gfCNCPoint4[21613] = {X 233.3038, Y 9.5049, Z -6.3333, A 0.000, B 0.000, C 0.000 }
gfCNCPoint4[21614] = {X 230.2485, Y 9.5049, Z -6.3333, A 0.000, B 0.000, C 0.000 }
gfCNCPoint4[21615] = {X 230.6107, Y 10.7176, Z -6.3333, A 0.000, B 0.000, C 0.000 }
gfCNCPoint4[21616] = {X 230.7574, Y 11.9748, Z -6.3333, A 0.000, B 0.000, C 0.000 }
gfCNCPoint4[21617] = {X 230.7597, Y 12.0808, Z -6.3333, A 0.000, B 0.000, C 0.000 }
gfCNCPoint4[21618] = {X 230.7605, Y 12.1868, Z -6.3333, A 0.000, B 0.000, C 0.000 }
gfCNCPoint4[21619] = {X 230.7602, Y 13.0462, Z -6.3333, A 0.000, B 0.000, C 0.000 }
gfCNCPoint4[21620] = {X 230.6532, Y 14.2233, Z -6.3333, A 0.000, B 0.000, C 0.000 }
gfCNCPoint4[21621] = {X 230.3572, Y 15.3675, Z -6.3333, A 0.000, B 0.000, C 0.000 }
gfCNCPoint4[21622] = {X 229.8799, Y 16.4488, Z -6.3333, A 0.000, B 0.000, C 0.000 }
gfCNCPoint4[21623] = {X 229.2339, Y 17.4386, Z -6.3333, A 0.000, B 0.000, C 0.000 }
gfCNCPoint4[21624] = {X 229.2342, Y 25.8570, Z -6.3333, A 0.000, B 0.000, C 0.000 }
gfCNCPoint4[21625] = {X 231.6342, Y 25.8569, Z -6.3333, A 0.000, B 0.000, C 0.000 }
gfCNCPoint4[21626] = {X 231.6347, Y 38.9924, Z -6.3333, A 0.000, B 0.000, C 0.000 }
gfCNCPoint4[21627] = {X 231.6440, Y 39.0069, Z -6.3333, A 0.000, B 0.000, C 0.000 }
gfCNCPoint4[21628] = {X 232.3931, Y 37.9855, Z -6.3333, A 0.000, B 0.000, C 0.000 }
gfCNCPoint4[21629] = {X 233.2692, Y 37.0706, Z -6.3333, A 0.000, B 0.000, C 0.000 }
gfCNCPoint4[21630] = {X 234.2573, Y 36.2780, Z -6.3333, A 0.000, B 0.000, C 0.000 }
gfCNCPoint4[21631] = {X 235.5691, Y 33.7103, Z -6.3333, A 0.000, B 0.000, C 0.000 }
gfCNCPoint4[21632] = {X 234.4282, Y 32.2860, Z -6.3333, A 0.000, B 0.000, C 0.000 }
gfCNCPoint4[21633] = {X 233.4498, Y 30.7456, Z -6.3333, A 0.000, B 0.000, C 0.000 }
gfCNCPoint4[21634] = {X 232.6455, Y 29.1076, Z -6.3333, A 0.000, B 0.000, C 0.000 }
gfCNCPoint4[21635] = {X 232.0249, Y 27.3915, Z -6.3333, A 0.000, B 0.000, C 0.000 }
gfCNCPoint4[21636] = {X 231.8157, Y 26.6277, Z -6.3333, A 0.000, B 0.000, C 0.000 }
gfCNCPoint4[21637] = {X 231.6342, Y 25.8569, Z -6.3333, A 0.000, B 0.000, C 0.000 }
gfCNCPoint4[21638] = {X 229.2342, Y 25.8570, Z -6.3333, A 0.000, B 0.000, C 0.000 }
gfCNCPoint4[21639] = {X 229.2347, Y 39.7493, Z -6.3333, A 0.000, B 0.000, C 0.000 }
gfCNCPoint4[21640] = {X 229.4337, Y 40.0185, Z -6.3333, A 0.000, B 0.000, C 0.000 }
gfCNCPoint4[21641] = {X 229.6200, Y 40.2966, Z -6.3333, A 0.000, B 0.000, C 0.000 }
gfCNCPoint4[21642] = {X 230.1055, Y 41.1910, Z -6.3333, A 0.000, B 0.000, C 0.000 }
gfCNCPoint4[21643] = {X 230.4616, Y 42.1443, Z -6.3333, A 0.000, B 0.000, C 0.000 }
gfCNCPoint4[21644] = {X 230.6813, Y 43.1379, Z -6.3333, A 0.000, B 0.000, C 0.000 }
gfCNCPoint4[21645] = {X 230.7603, Y 44.1524, Z -6.3333, A 0.000, B 0.000, C 0.000 }
gfCNCPoint4[21646] = {X 230.7605, Y 45.0000, Z -6.3333, A 0.000, B 0.000, C 0.000 }
gfCNCPoint4[21647] = {X 230.7459, Y 45.4609, Z -6.3333, A 0.000, B 0.000, C 0.000 }
gfCNCPoint4[21648] = {X 230.7021, Y 45.9200, Z -6.3333, A 0.000, B 0.000, C 0.000 }
gfCNCPoint4[21649] = {X 232.5859, Y 45.9200, Z -6.3333, A 0.000, B 0.000, C 0.000 }
gfCNCPoint4[21650] = {X 232.5421, Y 45.4609, Z -6.3333, A 0.000, B 0.000, C 0.000 }
gfCNCPoint4[21651] = {X 232.5275, Y 45.0000, Z -6.3333, A 0.000, B 0.000, C 0.000 }
gfCNCPoint4[21652] = {X 232.5275, Y 44.2089, Z -6.3333, A 0.000, B 0.000, C 0.000 }
gfCNCPoint4[21653] = {X 232.6006, Y 43.1798, Z -6.3333, A 0.000, B 0.000, C 0.000 }
gfCNCPoint4[21654] = {X 232.8184, Y 42.1714, Z -6.3333, A 0.000, B 0.000, C 0.000 }
gfCNCPoint4[21655] = {X 233.1766, Y 41.2038, Z -6.3333, A 0.000, B 0.000, C 0.000 }
gfCNCPoint4[21656] = {X 233.6680, Y 40.2966, Z -6.3333, A 0.000, B 0.000, C 0.000 }
gfCNCPoint4[21657] = {X 234.3527, Y 39.3876, Z -6.3333, A 0.000, B 0.000, C 0.000 }
gfCNCPoint4[21658] = {X 235.1707, Y 38.5964, Z -6.3333, A 0.000, B 0.000, C 0.000 }
gfCNCPoint4[21659] = {X 236.1021, Y 37.9424, Z -6.3333, A 0.000, B 0.000, C 0.000 }
gfCNCPoint4[21660] = {X 238.4997, Y 33.2492, Z -6.3333, A 0.000, B 0.000, C 0.000 }
gfCNCPoint4[21661] = {X 237.3859, Y 32.1414, Z -6.3333, A 0.000, B 0.000, C 0.000 }
gfCNCPoint4[21662] = {X 236.4005, Y 30.9179, Z -6.3333, A 0.000, B 0.000, C 0.000 }
gfCNCPoint4[21663] = {X 235.5554, Y 29.5936, Z -6.3333, A 0.000, B 0.000, C 0.000 }
gfCNCPoint4[21664] = {X 234.8609, Y 28.1845, Z -6.3333, A 0.000, B 0.000, C 0.000 }
gfCNCPoint4[21665] = {X 234.3254, Y 26.7076, Z -6.3333, A 0.000, B 0.000, C 0.000 }
gfCNCPoint4[21666] = {X 234.1405, Y 26.0316, Z -6.3333, A 0.000, B 0.000, C 0.000 }
gfCNCPoint4[21667] = {X 233.9799, Y 25.3493, Z -6.3333, A 0.000, B 0.000, C 0.000 }
gfCNCPoint4[21668] = {X 233.6672, Y 23.4597, Z -6.3333, A 0.000, B 0.000, C 0.000 }
gfCNCPoint4[21669] = {X 233.5414, Y 21.5485, Z -6.3333, A 0.000, B 0.000, C 0.000 }
gfCNCPoint4[21670] = {X 233.6038, Y 19.6342, Z -6.3333, A 0.000, B 0.000, C 0.000 }
gfCNCPoint4[21671] = {X 233.8537, Y 17.7353, Z -6.3333, A 0.000, B 0.000, C 0.000 }
gfCNCPoint4[21672] = {X 234.2887, Y 15.8701, Z -6.3333, A 0.000, B 0.000, C 0.000 }
gfCNCPoint4[21673] = {X 234.7349, Y 14.5420, Z -6.3333, A 0.000, B 0.000, C 0.000 }
gfCNCPoint4[21674] = {X 235.3045, Y 13.2620, Z -6.3333, A 0.000, B 0.000, C 0.000 }
gfCNCPoint4[21675] = {X 235.3657, Y 13.1418, Z -6.3333, A 0.000, B 0.000, C 0.000 }
gfCNCPoint4[21676] = {X 235.4279, Y 13.0222, Z -6.3333, A 0.000, B 0.000, C 0.000 }
gfCNCPoint4[21677] = {X 236.1692, Y 11.7670, Z -6.3333, A 0.000, B 0.000, C 0.000 }
gfCNCPoint4[21678] = {X 237.0303, Y 10.5908, Z -6.3333, A 0.000, B 0.000, C 0.000 }
gfCNCPoint4[21679] = {X 238.0029, Y 9.5049, Z -6.3333, A 0.000, B 0.000, C 0.000 }
gfCNCPoint4[21680] = {X 233.3038, Y 9.5049, Z -6.3333, A 0.000, B 0.000, C 0.000 }
gfCNCPoint4[21681] = {X 233.3038, Y 7.1049, Z -6.3333, A 0.000, B 0.000, C 0.000 }
gfCNCPoint4[21682] = {X 207.3611, Y 7.1049, Z -6.3333, A 0.000, B 0.000, C 0.000 }
gfCNCPoint4[21683] = {X 207.3611, Y 11.9049, Z -6.3333, A 0.000, B 0.000, C 0.000 }
gfCNCPoint4[21684] = {X 205.8579, Y 11.9049, Z -6.3333, A 0.000, B 0.000, C 0.000 }
gfCNCPoint4[21685] = {X 206.6129, Y 13.3419, Z -6.3333, A 0.000, B 0.000, C 0.000 }
gfCNCPoint4[21686] = {X 207.2383, Y 14.8398, Z -6.3333, A 0.000, B 0.000, C 0.000 }
gfCNCPoint4[21687] = {X 207.7991, Y 16.7126, Z -6.3333, A 0.000, B 0.000, C 0.000 }
gfCNCPoint4[21688] = {X 208.1779, Y 18.6305, Z -6.3333, A 0.000, B 0.000, C 0.000 }
gfCNCPoint4[21689] = {X 208.3712, Y 20.5759, Z -6.3333, A 0.000, B 0.000, C 0.000 }
gfCNCPoint4[21690] = {X 208.3773, Y 22.5308, Z -6.3333, A 0.000, B 0.000, C 0.000 }
gfCNCPoint4[21691] = {X 208.1960, Y 24.4773, Z -6.3333, A 0.000, B 0.000, C 0.000 }
gfCNCPoint4[21692] = {X 207.8292, Y 26.3975, Z -6.3333, A 0.000, B 0.000, C 0.000 }
gfCNCPoint4[21693] = {X 207.3620, Y 28.0101, Z -6.3333, A 0.000, B 0.000, C 0.000 }
gfCNCPoint4[21694] = {X 206.7385, Y 29.5690, Z -6.3333, A 0.000, B 0.000, C 0.000 }
gfCNCPoint4[21695] = {X 205.9648, Y 31.0590, Z -6.3333, A 0.000, B 0.000, C 0.000 }
gfCNCPoint4[21696] = {X 206.0466, Y 31.2168, Z -6.3333, A 0.000, B 0.000, C 0.000 }
gfCNCPoint4[21697] = {X 206.1255, Y 31.3760, Z -6.3333, A 0.000, B 0.000, C 0.000 }
gfCNCPoint4[21698] = {X 208.8842, Y 37.0755, Z -6.3333, A 0.000, B 0.000, C 0.000 }
gfCNCPoint4[21699] = {X 208.8842, Y 18.1966, Z -6.3333, A 0.000, B 0.000, C 0.000 }
gfCNCPoint4[21700] = {X 208.2325, Y 17.0008, Z -6.3333, A 0.000, B 0.000, C 0.000 }
gfCNCPoint4[21701] = {X 207.7551, Y 15.7254, Z -6.3333, A 0.000, B 0.000, C 0.000 }
gfCNCPoint4[21702] = {X 207.4614, Y 14.3956, Z -6.3333, A 0.000, B 0.000, C 0.000 }
gfCNCPoint4[21703] = {X 207.3572, Y 13.0378, Z -6.3333, A 0.000, B 0.000, C 0.000 }
gfCNCPoint4[21704] = {X 207.3570, Y 12.1868, Z -6.3333, A 0.000, B 0.000, C 0.000 }
gfCNCPoint4[21705] = {X 207.3580, Y 12.0458, Z -6.3333, A 0.000, B 0.000, C 0.000 }
gfCNCPoint4[21706] = {X 207.3611, Y 11.9049, Z -6.3333, A 0.000, B 0.000, C 0.000 }
gfCNCPoint4[21707] = {X 207.3611, Y 9.5049, Z -6.3333, A 0.000, B 0.000, C 0.000 }
gfCNCPoint4[21708] = {X 200.9085, Y 9.5049, Z -6.3333, A 0.000, B 0.000, C 0.000 }
gfCNCPoint4[21709] = {X 201.9821, Y 10.6133, Z -6.3333, A 0.000, B 0.000, C 0.000 }
gfCNCPoint4[21710] = {X 202.9438, Y 11.8201, Z -6.3333, A 0.000, B 0.000, C 0.000 }
gfCNCPoint4[21711] = {X 203.7847, Y 13.1140, Z -6.3333, A 0.000, B 0.000, C 0.000 }
gfCNCPoint4[21712] = {X 204.4380, Y 14.3567, Z -6.3333, A 0.000, B 0.000, C 0.000 }
gfCNCPoint4[21713] = {X 204.9798, Y 15.6519, Z -6.3333, A 0.000, B 0.000, C 0.000 }
gfCNCPoint4[21714] = {X 205.5523, Y 17.6384, Z -6.3333, A 0.000, B 0.000, C 0.000 }
gfCNCPoint4[21715] = {X 205.8929, Y 19.6775, Z -6.3333, A 0.000, B 0.000, C 0.000 }
gfCNCPoint4[21716] = {X 205.9974, Y 21.7422, Z -6.3333, A 0.000, B 0.000, C 0.000 }
gfCNCPoint4[21717] = {X 205.8641, Y 23.8052, Z -6.3333, A 0.000, B 0.000, C 0.000 }
gfCNCPoint4[21718] = {X 205.4950, Y 25.8393, Z -6.3333, A 0.000, B 0.000, C 0.000 }
gfCNCPoint4[21719] = {X 205.0938, Y 27.2257, Z -6.3333, A 0.000, B 0.000, C 0.000 }
gfCNCPoint4[21720] = {X 204.5582, Y 28.5659, Z -6.3333, A 0.000, B 0.000, C 0.000 }
gfCNCPoint4[21721] = {X 203.8933, Y 29.8469, Z -6.3333, A 0.000, B 0.000, C 0.000 }
gfCNCPoint4[21722] = {X 203.1057, Y 31.0563, Z -6.3333, A 0.000, B 0.000, C 0.000 }
gfCNCPoint4[21723] = {X 203.5734, Y 31.7151, Z -6.3333, A 0.000, B 0.000, C 0.000 }
gfCNCPoint4[21724] = {X 203.9653, Y 32.4217, Z -6.3333, A 0.000, B 0.000, C 0.000 }
gfCNCPoint4[21725] = {X 206.9865, Y 38.6634, Z -6.3333, A 0.000, B 0.000, C 0.000 }
gfCNCPoint4[21726] = {X 207.4240, Y 39.8017, Z -6.3333, A 0.000, B 0.000, C 0.000 }
gfCNCPoint4[21727] = {X 207.6653, Y 40.9971, Z -6.3333, A 0.000, B 0.000, C 0.000 }
gfCNCPoint4[21728] = {X 207.7038, Y 42.2159, Z -6.3333, A 0.000, B 0.000, C 0.000 }
gfCNCPoint4[21729] = {X 207.5382, Y 43.4241, Z -6.3333, A 0.000, B 0.000, C 0.000 }
gfCNCPoint4[21730] = {X 207.1733, Y 44.5877, Z -6.3333, A 0.000, B 0.000, C 0.000 }
gfCNCPoint4[21731] = {X 206.6193, Y 45.6741, Z -6.3333, A 0.000, B 0.000, C 0.000 }
gfCNCPoint4[21732] = {X 205.8917, Y 46.6527, Z -6.3333, A 0.000, B 0.000, C 0.000 }
gfCNCPoint4[21733] = {X 205.0110, Y 47.4962, Z -6.3333, A 0.000, B 0.000, C 0.000 }
gfCNCPoint4[21734] = {X 204.4751, Y 47.9295, Z -6.3333, A 0.000, B 0.000, C 0.000 }
gfCNCPoint4[21735] = {X 203.5896, Y 48.5433, Z -6.3333, A 0.000, B 0.000, C 0.000 }
gfCNCPoint4[21736] = {X 202.6234, Y 49.0199, Z -6.3333, A 0.000, B 0.000, C 0.000 }
gfCNCPoint4[21737] = {X 201.4894, Y 49.3740, Z -6.3333, A 0.000, B 0.000, C 0.000 }
gfCNCPoint4[21738] = {X 200.3130, Y 49.5392, Z -6.3333, A 0.000, B 0.000, C 0.000 }
gfCNCPoint4[21739] = {X 199.1253, Y 49.5112, Z -6.3333, A 0.000, B 0.000, C 0.000 }
gfCNCPoint4[21740] = {X 197.0993, Y 50.4925, Z -6.3333, A 0.000, B 0.000, C 0.000 }
gfCNCPoint4[21741] = {X 195.0081, Y 51.3261, Z -6.3333, A 0.000, B 0.000, C 0.000 }
gfCNCPoint4[21742] = {X 192.8625, Y 52.0075, Z -6.3333, A 0.000, B 0.000, C 0.000 }
gfCNCPoint4[21743] = {X 192.4425, Y 52.1234, Z -6.3333, A 0.000, B 0.000, C 0.000 }
gfCNCPoint4[21744] = {X 192.0206, Y 52.2321, Z -6.3333, A 0.000, B 0.000, C 0.000 }
gfCNCPoint4[21745] = {X 190.7204, Y 52.5192, Z -6.3333, A 0.000, B 0.000, C 0.000 }
gfCNCPoint4[21746] = {X 189.4070, Y 52.7376, Z -6.3333, A 0.000, B 0.000, C 0.000 }
gfCNCPoint4[21747] = {X 189.9007, Y 53.9117, Z -6.3333, A 0.000, B 0.000, C 0.000 }
gfCNCPoint4[21748] = {X 190.2679, Y 55.1313, Z -6.3333, A 0.000, B 0.000, C 0.000 }
gfCNCPoint4[21749] = {X 190.5268, Y 56.5553, Z -6.3333, A 0.000, B 0.000, C 0.000 }
gfCNCPoint4[21750] = {X 190.6135, Y 58.0000, Z -6.3333, A 0.000, B 0.000, C 0.000 }
gfCNCPoint4[21751] = {X 190.6132, Y 58.8756, Z -6.3333, A 0.000, B 0.000, C 0.000 }
gfCNCPoint4[21752] = {X 208.6248, Y 78.5343, Z -6.3333, A 0.000, B 0.000, C 0.000 }
gfCNCPoint4[21753] = {X 212.1639, Y 75.2917, Z -6.3333, A 0.000, B 0.000, C 0.000 }
gfCNCPoint4[21754] = {X 215.1986, Y 78.6038, Z -6.3333, A 0.000, B 0.000, C 0.000 }
gfCNCPoint4[21755] = {X 218.3263, Y 76.6002, Z -6.3333, A 0.000, B 0.000, C 0.000 }
gfCNCPoint4[21756] = {X 216.9980, Y 76.0790, Z -6.3333, A 0.000, B 0.000, C 0.000 }
gfCNCPoint4[21757] = {X 216.3745, Y 75.8855, Z -6.3333, A 0.000, B 0.000, C 0.000 }
gfCNCPoint4[21758] = {X 215.7268, Y 75.8033, Z -6.3333, A 0.000, B 0.000, C 0.000 }
gfCNCPoint4[21759] = {X 213.9317, Y 75.6427, Z -6.3333, A 0.000, B 0.000, C 0.000 }
gfCNCPoint4[21760] = {X 212.1639, Y 75.2917, Z -6.3333, A 0.000, B 0.000, C 0.000 }
gfCNCPoint4[21761] = {X 210.3944, Y 76.9130, Z -6.3333, A 0.000, B 0.000, C 0.000 }
gfCNCPoint4[21762] = {X 214.7930, Y 81.7139, Z -6.3333, A 0.000, B 0.000, C 0.000 }
gfCNCPoint4[21763] = {X 223.5811, Y 76.0841, Z -6.3333, A 0.000, B 0.000, C 0.000 }
gfCNCPoint4[21764] = {X 217.8868, Y 73.8496, Z -6.3333, A 0.000, B 0.000, C 0.000 }
gfCNCPoint4[21765] = {X 216.8707, Y 73.5373, Z -6.3333, A 0.000, B 0.000, C 0.000 }
gfCNCPoint4[21766] = {X 215.8159, Y 73.4049, Z -6.3333, A 0.000, B 0.000, C 0.000 }
gfCNCPoint4[21767] = {X 214.2744, Y 73.2673, Z -6.3333, A 0.000, B 0.000, C 0.000 }
gfCNCPoint4[21768] = {X 212.7564, Y 72.9660, Z -6.3333, A 0.000, B 0.000, C 0.000 }
gfCNCPoint4[21769] = {X 211.1573, Y 72.4583, Z -6.3333, A 0.000, B 0.000, C 0.000 }
gfCNCPoint4[21770] = {X 209.6276, Y 71.7691, Z -6.3333, A 0.000, B 0.000, C 0.000 }
gfCNCPoint4[21771] = {X 208.1879, Y 70.9075, Z -6.3333, A 0.000, B 0.000, C 0.000 }
gfCNCPoint4[21772] = {X 206.8576, Y 69.8853, Z -6.3333, A 0.000, B 0.000, C 0.000 }
gfCNCPoint4[21773] = {X 205.6544, Y 68.7159, Z -6.3333, A 0.000, B 0.000, C 0.000 }
gfCNCPoint4[21774] = {X 204.5946, Y 67.4153, Z -6.3333, A 0.000, B 0.000, C 0.000 }
gfCNCPoint4[21775] = {X 203.6923, Y 66.0008, Z -6.3333, A 0.000, B 0.000, C 0.000 }
gfCNCPoint4[21776] = {X 202.9597, Y 64.4914, Z -6.3333, A 0.000, B 0.000, C 0.000 }
gfCNCPoint4[21777] = {X 202.4066, Y 62.9075, Z -6.3333, A 0.000, B 0.000, C 0.000 }
gfCNCPoint4[21778] = {X 202.0405, Y 61.2701, Z -6.3333, A 0.000, B 0.000, C 0.000 }
gfCNCPoint4[21779] = {X 199.6719, Y 61.6573, Z -6.3333, A 0.000, B 0.000, C 0.000 }
gfCNCPoint4[21780] = {X 199.5094, Y 60.3398, Z -6.3333, A 0.000, B 0.000, C 0.000 }
gfCNCPoint4[21781] = {X 199.4510, Y 59.0136, Z -6.3333, A 0.000, B 0.000, C 0.000 }
gfCNCPoint4[21782] = {X 199.4508, Y 58.0000, Z -6.3333, A 0.000, B 0.000, C 0.000 }
gfCNCPoint4[21783] = {X 199.5411, Y 56.2566, Z -6.3333, A 0.000, B 0.000, C 0.000 }
gfCNCPoint4[21784] = {X 199.8109, Y 54.5319, Z -6.3333, A 0.000, B 0.000, C 0.000 }
gfCNCPoint4[21785] = {X 197.5976, Y 55.4819, Z -6.3333, A 0.000, B 0.000, C 0.000 }
gfCNCPoint4[21786] = {X 195.3259, Y 56.2825, Z -6.3333, A 0.000, B 0.000, C 0.000 }
gfCNCPoint4[21787] = {X 195.3577, Y 56.6287, Z -6.3333, A 0.000, B 0.000, C 0.000 }
gfCNCPoint4[21788] = {X 195.3824, Y 56.9755, Z -6.3333, A 0.000, B 0.000, C 0.000 }
gfCNCPoint4[21789] = {X 199.6719, Y 61.6573, Z -6.3333, A 0.000, B 0.000, C 0.000 }
gfCNCPoint4[21790] = {X 202.0405, Y 61.2701, Z -6.3333, A 0.000, B 0.000, C 0.000 }
gfCNCPoint4[21791] = {X 201.9013, Y 60.1424, Z -6.3333, A 0.000, B 0.000, C 0.000 }
gfCNCPoint4[21792] = {X 201.8510, Y 59.0073, Z -6.3333, A 0.000, B 0.000, C 0.000 }
gfCNCPoint4[21793] = {X 201.8508, Y 58.0000, Z -6.3333, A 0.000, B 0.000, C 0.000 }
gfCNCPoint4[21794] = {X 201.9282, Y 56.5045, Z -6.3333, A 0.000, B 0.000, C 0.000 }
gfCNCPoint4[21795] = {X 202.1597, Y 55.0250, Z -6.3333, A 0.000, B 0.000, C 0.000 }
gfCNCPoint4[21796] = {X 202.4964, Y 53.7245, Z -6.3333, A 0.000, B 0.000, C 0.000 }
gfCNCPoint4[21797] = {X 202.9522, Y 52.4609, Z -6.3333, A 0.000, B 0.000, C 0.000 }
gfCNCPoint4[21798] = {X 203.5231, Y 51.2449, Z -6.3333, A 0.000, B 0.000, C 0.000 }
gfCNCPoint4[21799] = {X 202.2638, Y 51.6564, Z -6.3333, A 0.000, B 0.000, C 0.000 }
gfCNCPoint4[21800] = {X 200.9603, Y 51.8923, Z -6.3333, A 0.000, B 0.000, C 0.000 }
gfCNCPoint4[21801] = {X 199.6367, Y 51.9482, Z -6.3333, A 0.000, B 0.000, C 0.000 }
gfCNCPoint4[21802] = {X 199.2155, Y 52.1566, Z -6.3333, A 0.000, B 0.000, C 0.000 }
gfCNCPoint4[21803] = {X 198.7914, Y 52.3592, Z -6.3333, A 0.000, B 0.000, C 0.000 }
gfCNCPoint4[21804] = {X 196.1934, Y 53.4485, Z -6.3333, A 0.000, B 0.000, C 0.000 }
gfCNCPoint4[21805] = {X 193.5136, Y 54.3175, Z -6.3333, A 0.000, B 0.000, C 0.000 }
gfCNCPoint4[21806] = {X 193.0575, Y 54.4433, Z -6.3333, A 0.000, B 0.000, C 0.000 }
gfCNCPoint4[21807] = {X 192.5993, Y 54.5613, Z -6.3333, A 0.000, B 0.000, C 0.000 }
gfCNCPoint4[21808] = {X 192.9061, Y 56.2397, Z -6.3333, A 0.000, B 0.000, C 0.000 }
gfCNCPoint4[21809] = {X 193.0134, Y 57.9426, Z -6.3333, A 0.000, B 0.000, C 0.000 }
gfCNCPoint4[21810] = {X 210.3944, Y 76.9130, Z -6.3333, A 0.000, B 0.000, C 0.000 }
gfCNCPoint4[21811] = {X 208.6248, Y 78.5343, Z -6.3333, A 0.000, B 0.000, C 0.000 }
gfCNCPoint4[21812] = {X 214.3875, Y 84.8240, Z -6.3333, A 0.000, B 0.000, C 0.000 }
gfCNCPoint4[21813] = {X 228.8358, Y 75.5680, Z -6.3333, A 0.000, B 0.000, C 0.000 }
gfCNCPoint4[21814] = {X 218.7736, Y 71.6194, Z -6.3333, A 0.000, B 0.000, C 0.000 }
gfCNCPoint4[21815] = {X 217.8428, Y 71.3053, Z -6.3333, A 0.000, B 0.000, C 0.000 }
gfCNCPoint4[21816] = {X 216.8820, Y 71.1001, Z -6.3333, A 0.000, B 0.000, C 0.000 }
gfCNCPoint4[21817] = {X 215.9041, Y 71.0065, Z -6.3333, A 0.000, B 0.000, C 0.000 }
gfCNCPoint4[21818] = {X 214.2345, Y 70.8308, Z -6.3333, A 0.000, B 0.000, C 0.000 }
gfCNCPoint4[21819] = {X 212.6054, Y 70.4253, Z -6.3333, A 0.000, B 0.000, C 0.000 }
gfCNCPoint4[21820] = {X 211.0482, Y 69.7978, Z -6.3333, A 0.000, B 0.000, C 0.000 }
gfCNCPoint4[21821] = {X 209.5931, Y 68.9605, Z -6.3333, A 0.000, B 0.000, C 0.000 }
gfCNCPoint4[21822] = {X 208.2681, Y 67.9296, Z -6.3333, A 0.000, B 0.000, C 0.000 }
gfCNCPoint4[21823] = {X 207.0988, Y 66.7249, Z -6.3333, A 0.000, B 0.000, C 0.000 }
gfCNCPoint4[21824] = {X 206.1079, Y 65.3697, Z -6.3333, A 0.000, B 0.000, C 0.000 }
gfCNCPoint4[21825] = {X 205.3143, Y 63.8903, Z -6.3333, A 0.000, B 0.000, C 0.000 }
gfCNCPoint4[21826] = {X 204.7336, Y 62.3151, Z -6.3333, A 0.000, B 0.000, C 0.000 }
gfCNCPoint4[21827] = {X 204.3768, Y 60.6746, Z -6.3333, A 0.000, B 0.000, C 0.000 }
gfCNCPoint4[21828] = {X 204.2510, Y 59.0005, Z -6.3333, A 0.000, B 0.000, C 0.000 }
gfCNCPoint4[21829] = {X 204.2508, Y 58.0000, Z -6.3333, A 0.000, B 0.000, C 0.000 }
gfCNCPoint4[21830] = {X 204.3396, Y 56.5378, Z -6.3333, A 0.000, B 0.000, C 0.000 }
gfCNCPoint4[21831] = {X 204.6048, Y 55.0972, Z -6.3333, A 0.000, B 0.000, C 0.000 }
gfCNCPoint4[21832] = {X 205.0423, Y 53.6992, Z -6.3333, A 0.000, B 0.000, C 0.000 }
gfCNCPoint4[21833] = {X 205.6459, Y 52.3645, Z -6.3333, A 0.000, B 0.000, C 0.000 }
gfCNCPoint4[21834] = {X 206.5294, Y 50.9389, Z -6.3333, A 0.000, B 0.000, C 0.000 }
gfCNCPoint4[21835] = {X 207.6019, Y 49.6494, Z -6.3333, A 0.000, B 0.000, C 0.000 }
gfCNCPoint4[21836] = {X 208.8426, Y 48.5209, Z -6.3333, A 0.000, B 0.000, C 0.000 }
gfCNCPoint4[21837] = {X 210.2277, Y 47.5751, Z -6.3333, A 0.000, B 0.000, C 0.000 }
gfCNCPoint4[21838] = {X 209.8801, Y 46.3328, Z -6.3333, A 0.000, B 0.000, C 0.000 }
gfCNCPoint4[21839] = {X 209.7572, Y 45.0487, Z -6.3333, A 0.000, B 0.000, C 0.000 }
gfCNCPoint4[21840] = {X 209.7570, Y 44.1918, Z -6.3333, A 0.000, B 0.000, C 0.000 }
gfCNCPoint4[21841] = {X 209.8558, Y 43.0029, Z -6.3333, A 0.000, B 0.000, C 0.000 }
gfCNCPoint4[21842] = {X 210.1495, Y 41.8467, Z -6.3333, A 0.000, B 0.000, C 0.000 }
gfCNCPoint4[21843] = {X 210.6300, Y 40.7548, Z -6.3333, A 0.000, B 0.000, C 0.000 }
gfCNCPoint4[21844] = {X 211.2842, Y 39.7572, Z -6.3333, A 0.000, B 0.000, C 0.000 }
gfCNCPoint4[21845] = {X 211.2842, Y 37.0755, Z -6.3333, A 0.000, B 0.000, C 0.000 }
gfCNCPoint4[21846] = {X 211.2839, Y 17.4390, Z -6.3333, A 0.000, B 0.000, C 0.000 }
gfCNCPoint4[21847] = {X 210.6358, Y 16.4454, Z -6.3333, A 0.000, B 0.000, C 0.000 }
gfCNCPoint4[21848] = {X 210.1576, Y 15.3597, Z -6.3333, A 0.000, B 0.000, C 0.000 }
gfCNCPoint4[21849] = {X 209.8621, Y 14.2108, Z -6.3333, A 0.000, B 0.000, C 0.000 }
gfCNCPoint4[21850] = {X 209.7572, Y 13.0291, Z -6.3333, A 0.000, B 0.000, C 0.000 }
gfCNCPoint4[21851] = {X 209.7570, Y 12.1868, Z -6.3333, A 0.000, B 0.000, C 0.000 }
gfCNCPoint4[21852] = {X 209.7578, Y 12.0808, Z -6.3333, A 0.000, B 0.000, C 0.000 }
gfCNCPoint4[21853] = {X 209.7601, Y 11.9748, Z -6.3333, A 0.000, B 0.000, C 0.000 }
gfCNCPoint4[21854] = {X 209.9068, Y 10.7176, Z -6.3333, A 0.000, B 0.000, C 0.000 }
gfCNCPoint4[21855] = {X 210.2690, Y 9.5049, Z -6.3333, A 0.000, B 0.000, C 0.000 }
gfCNCPoint4[21856] = {X 207.3611, Y 9.5049, Z -6.3333, A 0.000, B 0.000, C 0.000 }
gfCNCPoint4[21857] = {X 207.3611, Y 7.1049, Z -6.3333, A 0.000, B 0.000, C 0.000 }
gfCNCPoint4[21858] = {X 191.0955, Y 7.1049, Z -6.3333, A 0.000, B 0.000, C 0.000 }
gfCNCPoint4[21859] = {X 193.0686, Y 7.6379, Z -6.3333, A 0.000, B 0.000, C 0.000 }
gfCNCPoint4[21860] = {X 194.9670, Y 8.3953, Z -6.3333, A 0.000, B 0.000, C 0.000 }
gfCNCPoint4[21861] = {X 196.7651, Y 9.3670, Z -6.3333, A 0.000, B 0.000, C 0.000 }
gfCNCPoint4[21862] = {X 198.4389, Y 10.5400, Z -6.3333, A 0.000, B 0.000, C 0.000 }
gfCNCPoint4[21863] = {X 198.8603, Y 10.8896, Z -6.3333, A 0.000, B 0.000, C 0.000 }
gfCNCPoint4[21864] = {X 199.2672, Y 11.2559, Z -6.3333, A 0.000, B 0.000, C 0.000 }
gfCNCPoint4[21865] = {X 200.3523, Y 12.3983, Z -6.3333, A 0.000, B 0.000, C 0.000 }
gfCNCPoint4[21866] = {X 201.2979, Y 13.6587, Z -6.3333, A 0.000, B 0.000, C 0.000 }
gfCNCPoint4[21867] = {X 202.0911, Y 15.0200, Z -6.3333, A 0.000, B 0.000, C 0.000 }
gfCNCPoint4[21868] = {X 202.7214, Y 16.4641, Z -6.3333, A 0.000, B 0.000, C 0.000 }
gfCNCPoint4[21869] = {X 203.2150, Y 18.1838, Z -6.3333, A 0.000, B 0.000, C 0.000 }
gfCNCPoint4[21870] = {X 203.5083, Y 19.9487, Z -6.3333, A 0.000, B 0.000, C 0.000 }
gfCNCPoint4[21871] = {X 203.5973, Y 21.7356, Z -6.3333, A 0.000, B 0.000, C 0.000 }
gfCNCPoint4[21872] = {X 203.4810, Y 23.5209, Z -6.3333, A 0.000, B 0.000, C 0.000 }
gfCNCPoint4[21873] = {X 203.1608, Y 25.2812, Z -6.3333, A 0.000, B 0.000, C 0.000 }
gfCNCPoint4[21874] = {X 202.7603, Y 26.6266, Z -6.3333, A 0.000, B 0.000, C 0.000 }
gfCNCPoint4[21875] = {X 202.2086, Y 27.9174, Z -6.3333, A 0.000, B 0.000, C 0.000 }
gfCNCPoint4[21876] = {X 201.5130, Y 29.1367, Z -6.3333, A 0.000, B 0.000, C 0.000 }
gfCNCPoint4[21877] = {X 200.6824, Y 30.2684, Z -6.3333, A 0.000, B 0.000, C 0.000 }
gfCNCPoint4[21878] = {X 199.7279, Y 31.2977, Z -6.3333, A 0.000, B 0.000, C 0.000 }
gfCNCPoint4[21879] = {X 200.5671, Y 31.8701, Z -6.3333, A 0.000, B 0.000, C 0.000 }
gfCNCPoint4[21880] = {X 201.2697, Y 32.6039, Z -6.3333, A 0.000, B 0.000, C 0.000 }
gfCNCPoint4[21881] = {X 201.8050, Y 33.4673, Z -6.3333, A 0.000, B 0.000, C 0.000 }
gfCNCPoint4[21882] = {X 204.8262, Y 39.7091, Z -6.3333, A 0.000, B 0.000, C 0.000 }
gfCNCPoint4[21883] = {X 205.1508, Y 40.5847, Z -6.3333, A 0.000, B 0.000, C 0.000 }
gfCNCPoint4[21884] = {X 205.3026, Y 41.5062, Z -6.3333, A 0.000, B 0.000, C 0.000 }
gfCNCPoint4[21885] = {X 205.2761, Y 42.4397, Z -6.3333, A 0.000, B 0.000, C 0.000 }
gfCNCPoint4[21886] = {X 205.0723, Y 43.3511, Z -6.3333, A 0.000, B 0.000, C 0.000 }
gfCNCPoint4[21887] = {X 204.6986, Y 44.2070, Z -6.3333, A 0.000, B 0.000, C 0.000 }
gfCNCPoint4[21888] = {X 204.1687, Y 44.9760, Z -6.3333, A 0.000, B 0.000, C 0.000 }
gfCNCPoint4[21889] = {X 203.5020, Y 45.6299, Z -6.3333, A 0.000, B 0.000, C 0.000 }
gfCNCPoint4[21890] = {X 202.9659, Y 46.0634, Z -6.3333, A 0.000, B 0.000, C 0.000 }
gfCNCPoint4[21891] = {X 202.2141, Y 46.5642, Z -6.3333, A 0.000, B 0.000, C 0.000 }
gfCNCPoint4[21892] = {X 201.3829, Y 46.9182, Z -6.3333, A 0.000, B 0.000, C 0.000 }
gfCNCPoint4[21893] = {X 200.5008, Y 47.1133, Z -6.3333, A 0.000, B 0.000, C 0.000 }
gfCNCPoint4[21894] = {X 199.5979, Y 47.1427, Z -6.3333, A 0.000, B 0.000, C 0.000 }
gfCNCPoint4[21895] = {X 198.7050, Y 47.0056, Z -6.3333, A 0.000, B 0.000, C 0.000 }
gfCNCPoint4[21896] = {X 196.6156, Y 48.0776, Z -6.3333, A 0.000, B 0.000, C 0.000 }
gfCNCPoint4[21897] = {X 194.4463, Y 48.9769, Z -6.3333, A 0.000, B 0.000, C 0.000 }
gfCNCPoint4[21898] = {X 192.2113, Y 49.6975, Z -6.3333, A 0.000, B 0.000, C 0.000 }
gfCNCPoint4[21899] = {X 190.6550, Y 50.0838, Z -6.3333, A 0.000, B 0.000, C 0.000 }
gfCNCPoint4[21900] = {X 189.0755, Y 50.3606, Z -6.3333, A 0.000, B 0.000, C 0.000 }
gfCNCPoint4[21901] = {X 186.8993, Y 50.5591, Z -6.3333, A 0.000, B 0.000, C 0.000 }
gfCNCPoint4[21902] = {X 184.7140, Y 50.5499, Z -6.3333, A 0.000, B 0.000, C 0.000 }
gfCNCPoint4[21903] = {X 184.7389, Y 50.0706, Z -6.3333, A 0.000, B 0.000, C 0.000 }
gfCNCPoint4[21904] = {X 182.7586, Y 49.8798, Z -6.3333, A 0.000, B 0.000, C 0.000 }
gfCNCPoint4[21905] = {X 180.8029, Y 49.5148, Z -6.3333, A 0.000, B 0.000, C 0.000 }
gfCNCPoint4[21906] = {X 178.9540, Y 48.9789, Z -6.3333, A 0.000, B 0.000, C 0.000 }
gfCNCPoint4[21907] = {X 177.1792, Y 48.2334, Z -6.3333, A 0.000, B 0.000, C 0.000 }
gfCNCPoint4[21908] = {X 175.5022, Y 47.2883, Z -6.3333, A 0.000, B 0.000, C 0.000 }
gfCNCPoint4[21909] = {X 173.9453, Y 46.1562, Z -6.3333, A 0.000, B 0.000, C 0.000 }
gfCNCPoint4[21910] = {X 172.7970, Y 45.1084, Z -6.3333, A 0.000, B 0.000, C 0.000 }
gfCNCPoint4[21911] = {X 171.7809, Y 43.9320, Z -6.3333, A 0.000, B 0.000, C 0.000 }
gfCNCPoint4[21912] = {X 170.9111, Y 42.6435, Z -6.3333, A 0.000, B 0.000, C 0.000 }
gfCNCPoint4[21913] = {X 170.2001, Y 41.2611, Z -6.3333, A 0.000, B 0.000, C 0.000 }
gfCNCPoint4[21914] = {X 169.6577, Y 39.8043, Z -6.3333, A 0.000, B 0.000, C 0.000 }
gfCNCPoint4[21915] = {X 169.2916, Y 38.2935, Z -6.3333, A 0.000, B 0.000, C 0.000 }
gfCNCPoint4[21916] = {X 169.1811, Y 37.5991, Z -6.3333, A 0.000, B 0.000, C 0.000 }
gfCNCPoint4[21917] = {X 169.0220, Y 35.9859, Z -6.3333, A 0.000, B 0.000, C 0.000 }
gfCNCPoint4[21918] = {X 169.0392, Y 34.3649, Z -6.3333, A 0.000, B 0.000, C 0.000 }
gfCNCPoint4[21919] = {X 169.2323, Y 32.7554, Z -6.3333, A 0.000, B 0.000, C 0.000 }
gfCNCPoint4[21920] = {X 169.5992, Y 31.1764, Z -6.3333, A 0.000, B 0.000, C 0.000 }
gfCNCPoint4[21921] = {X 170.1354, Y 29.6466, Z -6.3333, A 0.000, B 0.000, C 0.000 }
gfCNCPoint4[21922] = {X 170.7623, Y 28.3590, Z -6.3333, A 0.000, B 0.000, C 0.000 }
gfCNCPoint4[21923] = {X 171.5520, Y 27.1643, Z -6.3333, A 0.000, B 0.000, C 0.000 }
gfCNCPoint4[21924] = {X 172.4911, Y 26.0830, Z -6.3333, A 0.000, B 0.000, C 0.000 }
gfCNCPoint4[21925] = {X 173.5635, Y 25.1338, Z -6.3333, A 0.000, B 0.000, C 0.000 }
gfCNCPoint4[21926] = {X 174.7507, Y 24.3328, Z -6.3333, A 0.000, B 0.000, C 0.000 }
gfCNCPoint4[21927] = {X 173.9908, Y 23.9225, Z -6.3333, A 0.000, B 0.000, C 0.000 }
gfCNCPoint4[21928] = {X 173.3256, Y 23.3716, Z -6.3333, A 0.000, B 0.000, C 0.000 }
gfCNCPoint4[21929] = {X 172.7809, Y 22.7015, Z -6.3333, A 0.000, B 0.000, C 0.000 }
gfCNCPoint4[21930] = {X 172.3776, Y 21.9378, Z -6.3333, A 0.000, B 0.000, C 0.000 }
gfCNCPoint4[21931] = {X 169.7664, Y 15.5423, Z -6.3333, A 0.000, B 0.000, C 0.000 }
gfCNCPoint4[21932] = {X 169.5125, Y 14.6752, Z -6.3333, A 0.000, B 0.000, C 0.000 }
gfCNCPoint4[21933] = {X 169.4412, Y 13.7745, Z -6.3333, A 0.000, B 0.000, C 0.000 }
gfCNCPoint4[21934] = {X 169.5553, Y 12.8782, Z -6.3333, A 0.000, B 0.000, C 0.000 }
gfCNCPoint4[21935] = {X 169.8501, Y 12.0241, Z -6.3333, A 0.000, B 0.000, C 0.000 }
gfCNCPoint4[21936] = {X 170.3131, Y 11.2482, Z -6.3333, A 0.000, B 0.000, C 0.000 }
gfCNCPoint4[21937] = {X 170.9249, Y 10.5833, Z -6.3333, A 0.000, B 0.000, C 0.000 }
gfCNCPoint4[21938] = {X 171.6596, Y 10.0573, Z -6.3333, A 0.000, B 0.000, C 0.000 }
gfCNCPoint4[21939] = {X 172.2916, Y 9.6970, Z -6.3333, A 0.000, B 0.000, C 0.000 }
gfCNCPoint4[21940] = {X 173.1774, Y 9.3226, Z -6.3333, A 0.000, B 0.000, C 0.000 }
gfCNCPoint4[21941] = {X 174.1234, Y 9.1497, Z -6.3333, A 0.000, B 0.000, C 0.000 }
gfCNCPoint4[21942] = {X 175.0843, Y 9.1863, Z -6.3333, A 0.000, B 0.000, C 0.000 }
gfCNCPoint4[21943] = {X 176.0143, Y 9.4309, Z -6.3333, A 0.000, B 0.000, C 0.000 }
gfCNCPoint4[21944] = {X 177.1159, Y 8.9623, Z -6.3333, A 0.000, B 0.000, C 0.000 }
gfCNCPoint4[21945] = {X 179.3009, Y 8.1586, Z -6.3333, A 0.000, B 0.000, C 0.000 }
gfCNCPoint4[21946] = {X 181.5549, Y 7.5759, Z -6.3333, A 0.000, B 0.000, C 0.000 }
gfCNCPoint4[21947] = {X 183.8557, Y 7.2200, Z -6.3333, A 0.000, B 0.000, C 0.000 }
gfCNCPoint4[21948] = {X 186.1804, Y 7.0943, Z -6.3333, A 0.000, B 0.000, C 0.000 }
gfCNCPoint4[21949] = {X 188.5061, Y 7.2003, Z -6.3333, A 0.000, B 0.000, C 0.000 }
gfCNCPoint4[21950] = {X 190.8098, Y 7.5367, Z -6.3333, A 0.000, B 0.000, C 0.000 }
gfCNCPoint4[21951] = {X 192.3918, Y 7.9275, Z -6.3333, A 0.000, B 0.000, C 0.000 }
gfCNCPoint4[21952] = {X 193.9295, Y 8.4665, Z -6.3333, A 0.000, B 0.000, C 0.000 }
gfCNCPoint4[21953] = {X 195.4093, Y 9.1487, Z -6.3333, A 0.000, B 0.000, C 0.000 }
gfCNCPoint4[21954] = {X 196.8178, Y 9.9681, Z -6.3333, A 0.000, B 0.000, C 0.000 }
gfCNCPoint4[21955] = {X 198.1423, Y 10.9173, Z -6.3333, A 0.000, B 0.000, C 0.000 }
gfCNCPoint4[21956] = {X 199.2090, Y 11.8667, Z -6.3333, A 0.000, B 0.000, C 0.000 }
gfCNCPoint4[21957] = {X 200.1662, Y 12.9264, Z -6.3333, A 0.000, B 0.000, C 0.000 }
gfCNCPoint4[21958] = {X 201.0023, Y 14.0840, Z -6.3333, A 0.000, B 0.000, C 0.000 }
gfCNCPoint4[21959] = {X 201.7075, Y 15.3258, Z -6.3333, A 0.000, B 0.000, C 0.000 }
gfCNCPoint4[21960] = {X 202.2734, Y 16.6369, Z -6.3333, A 0.000, B 0.000, C 0.000 }
gfCNCPoint4[21961] = {X 202.7496, Y 18.3014, Z -6.3333, A 0.000, B 0.000, C 0.000 }
gfCNCPoint4[21962] = {X 203.0321, Y 20.0095, Z -6.3333, A 0.000, B 0.000, C 0.000 }
gfCNCPoint4[21963] = {X 203.1173, Y 21.7387, Z -6.3333, A 0.000, B 0.000, C 0.000 }
gfCNCPoint4[21964] = {X 203.0041, Y 23.4663, Z -6.3333, A 0.000, B 0.000, C 0.000 }
gfCNCPoint4[21965] = {X 202.6939, Y 25.1696, Z -6.3333, A 0.000, B 0.000, C 0.000 }
gfCNCPoint4[21966] = {X 202.2592, Y 26.5986, Z -6.3333, A 0.000, B 0.000, C 0.000 }
gfCNCPoint4[21967] = {X 201.6470, Y 27.9611, Z -6.3333, A 0.000, B 0.000, C 0.000 }
gfCNCPoint4[21968] = {X 200.8672, Y 29.2351, Z -6.3333, A 0.000, B 0.000, C 0.000 }
gfCNCPoint4[21969] = {X 199.9325, Y 30.4002, Z -6.3333, A 0.000, B 0.000, C 0.000 }
gfCNCPoint4[21970] = {X 198.8578, Y 31.4375, Z -6.3333, A 0.000, B 0.000, C 0.000 }
gfCNCPoint4[21971] = {X 199.6407, Y 31.7993, Z -6.3333, A 0.000, B 0.000, C 0.000 }
gfCNCPoint4[21972] = {X 200.3380, Y 32.3069, Z -6.3333, A 0.000, B 0.000, C 0.000 }
gfCNCPoint4[21973] = {X 200.9229, Y 32.9407, Z -6.3333, A 0.000, B 0.000, C 0.000 }
gfCNCPoint4[21974] = {X 201.3730, Y 33.6764, Z -6.3333, A 0.000, B 0.000, C 0.000 }
gfCNCPoint4[21975] = {X 204.3942, Y 39.9182, Z -6.3333, A 0.000, B 0.000, C 0.000 }
gfCNCPoint4[21976] = {X 204.7207, Y 40.8441, Z -6.3333, A 0.000, B 0.000, C 0.000 }
gfCNCPoint4[21977] = {X 204.8337, Y 41.8194, Z -6.3333, A 0.000, B 0.000, C 0.000 }
gfCNCPoint4[21978] = {X 204.7276, Y 42.7955, Z -6.3333, A 0.000, B 0.000, C 0.000 }
gfCNCPoint4[21979] = {X 204.4078, Y 43.7238, Z -6.3333, A 0.000, B 0.000, C 0.000 }
gfCNCPoint4[21980] = {X 203.8900, Y 44.5580, Z -6.3333, A 0.000, B 0.000, C 0.000 }
gfCNCPoint4[21981] = {X 203.2002, Y 45.2567, Z -6.3333, A 0.000, B 0.000, C 0.000 }
gfCNCPoint4[21982] = {X 202.6641, Y 45.6901, Z -6.3333, A 0.000, B 0.000, C 0.000 }
gfCNCPoint4[21983] = {X 201.9528, Y 46.1596, Z -6.3333, A 0.000, B 0.000, C 0.000 }
gfCNCPoint4[21984] = {X 201.1645, Y 46.4835, Z -6.3333, A 0.000, B 0.000, C 0.000 }
gfCNCPoint4[21985] = {X 200.3287, Y 46.6497, Z -6.3333, A 0.000, B 0.000, C 0.000 }
gfCNCPoint4[21986] = {X 199.4764, Y 46.6520, Z -6.3333, A 0.000, B 0.000, C 0.000 }
gfCNCPoint4[21987] = {X 198.6397, Y 46.4904, Z -6.3333, A 0.000, B 0.000, C 0.000 }
gfCNCPoint4[21988] = {X 196.5324, Y 47.5869, Z -6.3333, A 0.000, B 0.000, C 0.000 }
gfCNCPoint4[21989] = {X 194.3411, Y 48.5040, Z -6.3333, A 0.000, B 0.000, C 0.000 }
gfCNCPoint4[21990] = {X 192.0811, Y 49.2355, Z -6.3333, A 0.000, B 0.000, C 0.000 }
gfCNCPoint4[21991] = {X 190.2777, Y 49.6712, Z -6.3333, A 0.000, B 0.000, C 0.000 }
gfCNCPoint4[21992] = {X 188.4445, Y 49.9567, Z -6.3333, A 0.000, B 0.000, C 0.000 }
gfCNCPoint4[21993] = {X 186.5940, Y 50.0901, Z -6.3333, A 0.000, B 0.000, C 0.000 }
gfCNCPoint4[21994] = {X 184.7389, Y 50.0706, Z -6.3333, A 0.000, B 0.000, C 0.000 }
gfCNCPoint4[21995] = {X 184.7140, Y 50.5499, Z -6.3333, A 0.000, B 0.000, C 0.000 }
gfCNCPoint4[21996] = {X 185.7095, Y 51.5033, Z -6.3333, A 0.000, B 0.000, C 0.000 }
gfCNCPoint4[21997] = {X 186.5595, Y 52.5883, Z -6.3333, A 0.000, B 0.000, C 0.000 }
gfCNCPoint4[21998] = {X 187.2467, Y 53.7831, Z -6.3333, A 0.000, B 0.000, C 0.000 }
gfCNCPoint4[21999] = {X 187.7797, Y 55.1348, Z -6.3333, A 0.000, B 0.000, C 0.000 }
gfCNCPoint4[22000] = {X 188.1044, Y 56.5511, Z -6.3333, A 0.000, B 0.000, C 0.000 }
gfCNCPoint4[22001] = {X 188.2135, Y 58.0000, Z -6.3333, A 0.000, B 0.000, C 0.000 }
gfCNCPoint4[22002] = {X 188.2132, Y 59.0140, Z -6.3333, A 0.000, B 0.000, C 0.000 }
gfCNCPoint4[22003] = {X 188.2027, Y 59.3922, Z -6.3333, A 0.000, B 0.000, C 0.000 }
gfCNCPoint4[22004] = {X 188.1774, Y 59.7697, Z -6.3333, A 0.000, B 0.000, C 0.000 }
gfCNCPoint4[22005] = {X 213.4317, Y 87.3334, Z -6.3333, A 0.000, B 0.000, C 0.000 }
gfCNCPoint4[22006] = {X 213.5229, Y 87.4312, Z -6.3333, A 0.000, B 0.000, C 0.000 }
gfCNCPoint4[22007] = {X 214.2179, Y 87.3787, Z -6.3333, A 0.000, B 0.000, C 0.000 }
gfCNCPoint4[22008] = {X 214.9136, Y 87.3372, Z -6.3333, A 0.000, B 0.000, C 0.000 }
gfCNCPoint4[22009] = {X 234.0906, Y 75.0519, Z -6.3333, A 0.000, B 0.000, C 0.000 }
gfCNCPoint4[22010] = {X 219.6591, Y 69.3887, Z -6.3333, A 0.000, B 0.000, C 0.000 }
gfCNCPoint4[22011] = {X 218.4692, Y 68.9885, Z -6.3333, A 0.000, B 0.000, C 0.000 }
gfCNCPoint4[22012] = {X 217.2413, Y 68.7271, Z -6.3333, A 0.000, B 0.000, C 0.000 }
gfCNCPoint4[22013] = {X 215.9916, Y 68.6081, Z -6.3333, A 0.000, B 0.000, C 0.000 }
gfCNCPoint4[22014] = {X 214.5215, Y 68.4435, Z -6.3333, A 0.000, B 0.000, C 0.000 }
gfCNCPoint4[22015] = {X 213.0937, Y 68.0568, Z -6.3333, A 0.000, B 0.000, C 0.000 }
gfCNCPoint4[22016] = {X 211.7415, Y 67.4570, Z -6.3333, A 0.000, B 0.000, C 0.000 }
gfCNCPoint4[22017] = {X 210.4964, Y 66.6582, Z -6.3333, A 0.000, B 0.000, C 0.000 }
gfCNCPoint4[22018] = {X 209.3876, Y 65.6790, Z -6.3333, A 0.000, B 0.000, C 0.000 }
gfCNCPoint4[22019] = {X 208.4409, Y 64.5423, Z -6.3333, A 0.000, B 0.000, C 0.000 }
gfCNCPoint4[22020] = {X 207.6785, Y 63.2747, Z -6.3333, A 0.000, B 0.000, C 0.000 }
gfCNCPoint4[22021] = {X 207.1182, Y 61.9056, Z -6.3333, A 0.000, B 0.000, C 0.000 }
gfCNCPoint4[22022] = {X 206.7730, Y 60.4672, Z -6.3333, A 0.000, B 0.000, C 0.000 }
gfCNCPoint4[22023] = {X 206.6510, Y 58.9930, Z -6.3333, A 0.000, B 0.000, C 0.000 }
gfCNCPoint4[22024] = {X 206.6508, Y 58.0000, Z -6.3333, A 0.000, B 0.000, C 0.000 }
gfCNCPoint4[22025] = {X 206.7577, Y 56.5655, Z -6.3333, A 0.000, B 0.000, C 0.000 }
gfCNCPoint4[22026] = {X 207.0760, Y 55.1628, Z -6.3333, A 0.000, B 0.000, C 0.000 }
gfCNCPoint4[22027] = {X 207.5986, Y 53.8226, Z -6.3333, A 0.000, B 0.000, C 0.000 }
gfCNCPoint4[22028] = {X 208.3140, Y 52.5747, Z -6.3333, A 0.000, B 0.000, C 0.000 }
gfCNCPoint4[22029] = {X 209.2065, Y 51.4466, Z -6.3333, A 0.000, B 0.000, C 0.000 }
gfCNCPoint4[22030] = {X 210.2563, Y 50.4632, Z -6.3333, A 0.000, B 0.000, C 0.000 }
gfCNCPoint4[22031] = {X 211.4402, Y 49.6463, Z -6.3333, A 0.000, B 0.000, C 0.000 }
gfCNCPoint4[22032] = {X 212.5893, Y 49.0723, Z -6.3333, A 0.000, B 0.000, C 0.000 }
gfCNCPoint4[22033] = {X 213.8042, Y 48.6556, Z -6.3333, A 0.000, B 0.000, C 0.000 }
gfCNCPoint4[22034] = {X 213.2578, Y 48.0874, Z -6.3333, A 0.000, B 0.000, C 0.000 }
gfCNCPoint4[22035] = {X 212.8100, Y 47.4386, Z -6.3333, A 0.000, B 0.000, C 0.000 }
gfCNCPoint4[22036] = {X 212.4725, Y 46.7262, Z -6.3333, A 0.000, B 0.000, C 0.000 }
gfCNCPoint4[22037] = {X 212.2401, Y 45.8965, Z -6.3333, A 0.000, B 0.000, C 0.000 }
gfCNCPoint4[22038] = {X 212.1572, Y 45.0389, Z -6.3333, A 0.000, B 0.000, C 0.000 }
gfCNCPoint4[22039] = {X 212.1570, Y 44.1918, Z -6.3333, A 0.000, B 0.000, C 0.000 }
gfCNCPoint4[22040] = {X 212.2382, Y 43.3126, Z -6.3333, A 0.000, B 0.000, C 0.000 }
gfCNCPoint4[22041] = {X 212.4789, Y 42.4632, Z -6.3333, A 0.000, B 0.000, C 0.000 }
gfCNCPoint4[22042] = {X 212.8711, Y 41.6722, Z -6.3333, A 0.000, B 0.000, C 0.000 }
gfCNCPoint4[22043] = {X 213.4015, Y 40.9663, Z -6.3333, A 0.000, B 0.000, C 0.000 }
gfCNCPoint4[22044] = {X 213.6815, Y 40.6575, Z -6.3333, A 0.000, B 0.000, C 0.000 }
gfCNCPoint4[22045] = {X 213.6842, Y 40.3040, Z -6.3333, A 0.000, B 0.000, C 0.000 }
gfCNCPoint4[22046] = {X 213.6842, Y 17.4646, Z -6.3333, A 0.000, B 0.000, C 0.000 }
gfCNCPoint4[22047] = {X 213.6789, Y 16.7696, Z -6.3333, A 0.000, B 0.000, C 0.000 }
gfCNCPoint4[22048] = {X 213.6786, Y 16.5186, Z -6.3333, A 0.000, B 0.000, C 0.000 }
gfCNCPoint4[22049] = {X 213.0398, Y 15.7774, Z -6.3333, A 0.000, B 0.000, C 0.000 }
gfCNCPoint4[22050] = {X 212.5616, Y 14.9236, Z -6.3333, A 0.000, B 0.000, C 0.000 }
gfCNCPoint4[22051] = {X 212.2634, Y 13.9916, Z -6.3333, A 0.000, B 0.000, C 0.000 }
gfCNCPoint4[22052] = {X 212.1572, Y 13.0188, Z -6.3333, A 0.000, B 0.000, C 0.000 }
gfCNCPoint4[22053] = {X 212.1570, Y 12.1868, Z -6.3333, A 0.000, B 0.000, C 0.000 }
gfCNCPoint4[22054] = {X 212.2436, Y 11.2717, Z -6.3333, A 0.000, B 0.000, C 0.000 }
gfCNCPoint4[22055] = {X 212.5002, Y 10.3890, Z -6.3333, A 0.000, B 0.000, C 0.000 }
gfCNCPoint4[22056] = {X 212.9449, Y 9.5280, Z -6.3333, A 0.000, B 0.000, C 0.000 }
gfCNCPoint4[22057] = {X 213.5511, Y 8.7718, Z -6.3333, A 0.000, B 0.000, C 0.000 }
gfCNCPoint4[22058] = {X 214.2946, Y 8.1503, Z -6.3333, A 0.000, B 0.000, C 0.000 }
gfCNCPoint4[22059] = {X 215.1464, Y 7.6879, Z -6.3333, A 0.000, B 0.000, C 0.000 }
gfCNCPoint4[22060] = {X 216.0727, Y 7.4030, Z -6.3333, A 0.000, B 0.000, C 0.000 }
gfCNCPoint4[22061] = {X 217.0370, Y 7.3068, Z -6.3333, A 0.000, B 0.000, C 0.000 }
gfCNCPoint4[22062] = {X 223.4805, Y 7.3068, Z -6.3333, A 0.000, B 0.000, C 0.000 }
gfCNCPoint4[22063] = {X 224.4448, Y 7.4030, Z -6.3333, A 0.000, B 0.000, C 0.000 }
gfCNCPoint4[22064] = {X 225.3711, Y 7.6879, Z -6.3333, A 0.000, B 0.000, C 0.000 }
gfCNCPoint4[22065] = {X 226.2229, Y 8.1503, Z -6.3333, A 0.000, B 0.000, C 0.000 }
gfCNCPoint4[22066] = {X 226.9664, Y 8.7718, Z -6.3333, A 0.000, B 0.000, C 0.000 }
gfCNCPoint4[22067] = {X 227.5726, Y 9.5280, Z -6.3333, A 0.000, B 0.000, C 0.000 }
gfCNCPoint4[22068] = {X 228.0173, Y 10.3890, Z -6.3333, A 0.000, B 0.000, C 0.000 }
gfCNCPoint4[22069] = {X 228.2739, Y 11.2717, Z -6.3333, A 0.000, B 0.000, C 0.000 }
gfCNCPoint4[22070] = {X 228.3605, Y 12.1868, Z -6.3333, A 0.000, B 0.000, C 0.000 }
gfCNCPoint4[22071] = {X 228.3603, Y 13.0237, Z -6.3333, A 0.000, B 0.000, C 0.000 }
gfCNCPoint4[22072] = {X 228.2529, Y 13.9969, Z -6.3333, A 0.000, B 0.000, C 0.000 }
gfCNCPoint4[22073] = {X 227.9535, Y 14.9290, Z -6.3333, A 0.000, B 0.000, C 0.000 }
gfCNCPoint4[22074] = {X 227.4741, Y 15.7826, Z -6.3333, A 0.000, B 0.000, C 0.000 }
gfCNCPoint4[22075] = {X 226.8339, Y 16.5233, Z -6.3333, A 0.000, B 0.000, C 0.000 }
gfCNCPoint4[22076] = {X 226.8348, Y 40.6643, Z -6.3333, A 0.000, B 0.000, C 0.000 }
gfCNCPoint4[22077] = {X 227.4747, Y 41.4051, Z -6.3333, A 0.000, B 0.000, C 0.000 }
gfCNCPoint4[22078] = {X 227.9539, Y 42.2587, Z -6.3333, A 0.000, B 0.000, C 0.000 }
gfCNCPoint4[22079] = {X 228.2531, Y 43.1908, Z -6.3333, A 0.000, B 0.000, C 0.000 }
gfCNCPoint4[22080] = {X 228.3603, Y 44.1638, Z -6.3333, A 0.000, B 0.000, C 0.000 }
gfCNCPoint4[22081] = {X 228.3605, Y 45.0000, Z -6.3333, A 0.000, B 0.000, C 0.000 }
gfCNCPoint4[22082] = {X 228.3507, Y 45.3090, Z -6.3333, A 0.000, B 0.000, C 0.000 }
gfCNCPoint4[22083] = {X 228.3214, Y 45.6167, Z -6.3333, A 0.000, B 0.000, C 0.000 }
gfCNCPoint4[22084] = {X 228.0910, Y 46.5992, Z -6.3333, A 0.000, B 0.000, C 0.000 }
gfCNCPoint4[22085] = {X 227.6635, Y 47.5134, Z -6.3333, A 0.000, B 0.000, C 0.000 }
gfCNCPoint4[22086] = {X 227.0571, Y 48.3200, Z -6.3333, A 0.000, B 0.000, C 0.000 }
gfCNCPoint4[22087] = {X 226.7053, Y 47.9934, Z -6.3333, A 0.000, B 0.000, C 0.000 }
gfCNCPoint4[22088] = {X 226.0261, Y 48.5889, Z -6.3333, A 0.000, B 0.000, C 0.000 }
gfCNCPoint4[22089] = {X 225.2396, Y 49.0331, Z -6.3333, A 0.000, B 0.000, C 0.000 }
gfCNCPoint4[22090] = {X 224.3790, Y 49.3073, Z -6.3333, A 0.000, B 0.000, C 0.000 }
gfCNCPoint4[22091] = {X 223.4805, Y 49.4000, Z -6.3333, A 0.000, B 0.000, C 0.000 }
gfCNCPoint4[22092] = {X 217.0370, Y 49.4000, Z -6.3333, A 0.000, B 0.000, C 0.000 }
gfCNCPoint4[22093] = {X 216.0579, Y 49.2897, Z -6.3333, A 0.000, B 0.000, C 0.000 }
gfCNCPoint4[22094] = {X 215.1279, Y 48.9643, Z -6.3333, A 0.000, B 0.000, C 0.000 }
gfCNCPoint4[22095] = {X 214.2937, Y 48.4400, Z -6.3333, A 0.000, B 0.000, C 0.000 }
gfCNCPoint4[22096] = {X 213.5969, Y 47.7433, Z -6.3333, A 0.000, B 0.000, C 0.000 }
gfCNCPoint4[22097] = {X 213.0727, Y 46.9091, Z -6.3333, A 0.000, B 0.000, C 0.000 }
gfCNCPoint4[22098] = {X 212.7473, Y 45.9791, Z -6.3333, A 0.000, B 0.000, C 0.000 }
gfCNCPoint4[22099] = {X 212.6370, Y 45.0000, Z -6.3333, A 0.000, B 0.000, C 0.000 }
gfCNCPoint4[22100] = {X 212.6370, Y 44.1918, Z -6.3333, A 0.000, B 0.000, C 0.000 }
gfCNCPoint4[22101] = {X 212.7101, Y 43.4005, Z -6.3333, A 0.000, B 0.000, C 0.000 }
gfCNCPoint4[22102] = {X 212.9267, Y 42.6360, Z -6.3333, A 0.000, B 0.000, C 0.000 }
gfCNCPoint4[22103] = {X 213.2797, Y 41.9240, Z -6.3333, A 0.000, B 0.000, C 0.000 }
gfCNCPoint4[22104] = {X 213.7571, Y 41.2887, Z -6.3333, A 0.000, B 0.000, C 0.000 }
gfCNCPoint4[22105] = {X 214.1601, Y 40.8442, Z -6.3333, A 0.000, B 0.000, C 0.000 }
gfCNCPoint4[22106] = {X 214.1642, Y 40.3060, Z -6.3333, A 0.000, B 0.000, C 0.000 }
gfCNCPoint4[22107] = {X 214.1642, Y 17.4626, Z -6.3333, A 0.000, B 0.000, C 0.000 }
gfCNCPoint4[22108] = {X 214.1589, Y 16.7691, Z -6.3333, A 0.000, B 0.000, C 0.000 }
gfCNCPoint4[22109] = {X 214.1584, Y 16.3058, Z -6.3333, A 0.000, B 0.000, C 0.000 }
gfCNCPoint4[22110] = {X 213.5163, Y 15.6171, Z -6.3333, A 0.000, B 0.000, C 0.000 }
gfCNCPoint4[22111] = {X 213.0354, Y 14.8075, Z -6.3333, A 0.000, B 0.000, C 0.000 }
gfCNCPoint4[22112] = {X 212.7378, Y 13.9142, Z -6.3333, A 0.000, B 0.000, C 0.000 }
gfCNCPoint4[22113] = {X 212.6370, Y 12.9780, Z -6.3333, A 0.000, B 0.000, C 0.000 }
gfCNCPoint4[22114] = {X 212.6370, Y 12.1868, Z -6.3333, A 0.000, B 0.000, C 0.000 }
gfCNCPoint4[22115] = {X 212.7473, Y 11.2077, Z -6.3333, A 0.000, B 0.000, C 0.000 }
gfCNCPoint4[22116] = {X 213.0728, Y 10.2777, Z -6.3333, A 0.000, B 0.000, C 0.000 }
gfCNCPoint4[22117] = {X 213.5970, Y 9.4435, Z -6.3333, A 0.000, B 0.000, C 0.000 }
gfCNCPoint4[22118] = {X 214.2937, Y 8.7468, Z -6.3333, A 0.000, B 0.000, C 0.000 }
gfCNCPoint4[22119] = {X 215.1279, Y 8.2226, Z -6.3333, A 0.000, B 0.000, C 0.000 }
gfCNCPoint4[22120] = {X 216.0579, Y 7.8971, Z -6.3333, A 0.000, B 0.000, C 0.000 }
gfCNCPoint4[22121] = {X 217.0370, Y 7.7868, Z -6.3333, A 0.000, B 0.000, C 0.000 }
gfCNCPoint4[22122] = {X 223.4805, Y 7.7868, Z -6.3333, A 0.000, B 0.000, C 0.000 }
gfCNCPoint4[22123] = {X 224.4596, Y 7.8971, Z -6.3333, A 0.000, B 0.000, C 0.000 }
gfCNCPoint4[22124] = {X 225.3896, Y 8.2226, Z -6.3333, A 0.000, B 0.000, C 0.000 }
gfCNCPoint4[22125] = {X 226.2238, Y 8.7468, Z -6.3333, A 0.000, B 0.000, C 0.000 }
gfCNCPoint4[22126] = {X 226.9205, Y 9.4435, Z -6.3333, A 0.000, B 0.000, C 0.000 }
gfCNCPoint4[22127] = {X 227.4447, Y 10.2777, Z -6.3333, A 0.000, B 0.000, C 0.000 }
gfCNCPoint4[22128] = {X 227.7702, Y 11.2077, Z -6.3333, A 0.000, B 0.000, C 0.000 }
gfCNCPoint4[22129] = {X 227.8805, Y 12.1868, Z -6.3333, A 0.000, B 0.000, C 0.000 }
gfCNCPoint4[22130] = {X 227.8802, Y 13.0233, Z -6.3333, A 0.000, B 0.000, C 0.000 }
gfCNCPoint4[22131] = {X 227.7720, Y 13.9491, Z -6.3333, A 0.000, B 0.000, C 0.000 }
gfCNCPoint4[22132] = {X 227.4712, Y 14.8312, Z -6.3333, A 0.000, B 0.000, C 0.000 }
gfCNCPoint4[22133] = {X 226.9913, Y 15.6303, Z -6.3333, A 0.000, B 0.000, C 0.000 }
gfCNCPoint4[22134] = {X 226.3538, Y 16.3103, Z -6.3333, A 0.000, B 0.000, C 0.000 }
gfCNCPoint4[22135] = {X 226.3548, Y 40.8774, Z -6.3333, A 0.000, B 0.000, C 0.000 }
gfCNCPoint4[22136] = {X 226.9987, Y 41.5664, Z -6.3333, A 0.000, B 0.000, C 0.000 }
gfCNCPoint4[22137] = {X 227.4809, Y 42.3767, Z -6.3333, A 0.000, B 0.000, C 0.000 }
gfCNCPoint4[22138] = {X 227.7794, Y 43.2713, Z -6.3333, A 0.000, B 0.000, C 0.000 }
gfCNCPoint4[22139] = {X 227.8805, Y 44.2089, Z -6.3333, A 0.000, B 0.000, C 0.000 }
gfCNCPoint4[22140] = {X 227.8805, Y 45.0000, Z -6.3333, A 0.000, B 0.000, C 0.000 }
gfCNCPoint4[22141] = {X 227.8037, Y 45.8182, Z -6.3333, A 0.000, B 0.000, C 0.000 }
gfCNCPoint4[22142] = {X 227.5762, Y 46.6079, Z -6.3333, A 0.000, B 0.000, C 0.000 }
gfCNCPoint4[22143] = {X 227.2057, Y 47.3415, Z -6.3333, A 0.000, B 0.000, C 0.000 }
gfCNCPoint4[22144] = {X 226.7053, Y 47.9934, Z -6.3333, A 0.000, B 0.000, C 0.000 }
gfCNCPoint4[22145] = {X 227.0571, Y 48.3200, Z -6.3333, A 0.000, B 0.000, C 0.000 }
gfCNCPoint4[22146] = {X 236.2309, Y 48.3200, Z -6.3333, A 0.000, B 0.000, C 0.000 }
gfCNCPoint4[22147] = {X 235.6245, Y 47.5134, Z -6.3333, A 0.000, B 0.000, C 0.000 }
gfCNCPoint4[22148] = {X 235.1970, Y 46.5992, Z -6.3333, A 0.000, B 0.000, C 0.000 }
gfCNCPoint4[22149] = {X 234.9666, Y 45.6167, Z -6.3333, A 0.000, B 0.000, C 0.000 }
gfCNCPoint4[22150] = {X 234.9373, Y 45.3090, Z -6.3333, A 0.000, B 0.000, C 0.000 }
gfCNCPoint4[22151] = {X 234.9275, Y 45.0000, Z -6.3333, A 0.000, B 0.000, C 0.000 }
gfCNCPoint4[22152] = {X 234.9275, Y 44.2089, Z -6.3333, A 0.000, B 0.000, C 0.000 }
gfCNCPoint4[22153] = {X 235.0194, Y 43.2661, Z -6.3333, A 0.000, B 0.000, C 0.000 }
gfCNCPoint4[22154] = {X 235.2918, Y 42.3588, Z -6.3333, A 0.000, B 0.000, C 0.000 }
gfCNCPoint4[22155] = {X 235.7342, Y 41.5212, Z -6.3333, A 0.000, B 0.000, C 0.000 }
gfCNCPoint4[22156] = {X 236.3302, Y 40.7849, Z -6.3333, A 0.000, B 0.000, C 0.000 }
gfCNCPoint4[22157] = {X 237.0572, Y 40.1776, Z -6.3333, A 0.000, B 0.000, C 0.000 }
gfCNCPoint4[22158] = {X 237.8878, Y 39.7222, Z -6.3333, A 0.000, B 0.000, C 0.000 }
gfCNCPoint4[22159] = {X 241.5461, Y 32.5615, Z -6.3333, A 0.000, B 0.000, C 0.000 }
gfCNCPoint4[22160] = {X 240.2116, Y 31.5587, Z -6.3333, A 0.000, B 0.000, C 0.000 }
gfCNCPoint4[22161] = {X 239.0307, Y 30.3787, Z -6.3333, A 0.000, B 0.000, C 0.000 }
gfCNCPoint4[22162] = {X 238.0270, Y 29.0449, Z -6.3333, A 0.000, B 0.000, C 0.000 }
gfCNCPoint4[22163] = {X 237.2200, Y 27.5836, Z -6.3333, A 0.000, B 0.000, C 0.000 }
gfCNCPoint4[22164] = {X 236.6259, Y 26.0235, Z -6.3333, A 0.000, B 0.000, C 0.000 }
gfCNCPoint4[22165] = {X 236.1908, Y 24.1499, Z -6.3333, A 0.000, B 0.000, C 0.000 }
gfCNCPoint4[22166] = {X 235.9688, Y 22.2393, Z -6.3333, A 0.000, B 0.000, C 0.000 }
gfCNCPoint4[22167] = {X 235.9630, Y 20.3158, Z -6.3333, A 0.000, B 0.000, C 0.000 }
gfCNCPoint4[22168] = {X 236.1732, Y 18.4038, Z -6.3333, A 0.000, B 0.000, C 0.000 }
gfCNCPoint4[22169] = {X 236.5969, Y 16.5276, Z -6.3333, A 0.000, B 0.000, C 0.000 }
gfCNCPoint4[22170] = {X 237.1163, Y 15.0570, Z -6.3333, A 0.000, B 0.000, C 0.000 }
gfCNCPoint4[22171] = {X 237.8160, Y 13.6631, Z -6.3333, A 0.000, B 0.000, C 0.000 }
gfCNCPoint4[22172] = {X 238.6851, Y 12.3680, Z -6.3333, A 0.000, B 0.000, C 0.000 }
gfCNCPoint4[22173] = {X 239.7097, Y 11.1922, Z -6.3333, A 0.000, B 0.000, C 0.000 }
gfCNCPoint4[22174] = {X 240.8741, Y 10.1539, Z -6.3333, A 0.000, B 0.000, C 0.000 }
gfCNCPoint4[22175] = {X 242.1595, Y 9.2698, Z -6.3333, A 0.000, B 0.000, C 0.000 }
gfCNCPoint4[22176] = {X 243.5458, Y 8.5541, Z -6.3333, A 0.000, B 0.000, C 0.000 }
gfCNCPoint4[22177] = {X 245.0108, Y 8.0179, Z -6.3333, A 0.000, B 0.000, C 0.000 }
gfCNCPoint4[22178] = {X 246.5316, Y 7.6698, Z -6.3333, A 0.000, B 0.000, C 0.000 }
gfCNCPoint4[22179] = {X 248.6761, Y 7.3923, Z -6.3333, A 0.000, B 0.000, C 0.000 }
gfCNCPoint4[22180] = {X 250.8369, Y 7.3099, Z -6.3333, A 0.000, B 0.000, C 0.000 }
gfCNCPoint4[22181] = {X 266.7608, Y 7.3099, Z -6.3333, A 0.000, B 0.000, C 0.000 }
gfCNCPoint4[22182] = {X 267.7192, Y 7.4113, Z -6.3333, A 0.000, B 0.000, C 0.000 }
gfCNCPoint4[22183] = {X 268.6389, Y 7.6990, Z -6.3333, A 0.000, B 0.000, C 0.000 }
gfCNCPoint4[22184] = {X 269.4843, Y 8.1618, Z -6.3333, A 0.000, B 0.000, C 0.000 }
gfCNCPoint4[22185] = {X 270.2223, Y 8.7816, Z -6.3333, A 0.000, B 0.000, C 0.000 }
gfCNCPoint4[22186] = {X 270.8242, Y 9.5343, Z -6.3333, A 0.000, B 0.000, C 0.000 }
gfCNCPoint4[22187] = {X 271.2665, Y 10.3905, Z -6.3333, A 0.000, B 0.000, C 0.000 }
gfCNCPoint4[22188] = {X 271.5235, Y 11.2718, Z -6.3333, A 0.000, B 0.000, C 0.000 }
gfCNCPoint4[22189] = {X 271.6110, Y 12.1857, Z -6.3333, A 0.000, B 0.000, C 0.000 }
gfCNCPoint4[22190] = {X 271.6108, Y 13.0237, Z -6.3333, A 0.000, B 0.000, C 0.000 }
gfCNCPoint4[22191] = {X 271.5128, Y 13.9524, Z -6.3333, A 0.000, B 0.000, C 0.000 }
gfCNCPoint4[22192] = {X 271.2396, Y 14.8453, Z -6.3333, A 0.000, B 0.000, C 0.000 }
gfCNCPoint4[22193] = {X 275.6743, Y 16.6820, Z -6.3333, A 0.000, B 0.000, C 0.000 }
gfCNCPoint4[22194] = {X 275.3129, Y 17.4562, Z -6.3333, A 0.000, B 0.000, C 0.000 }
gfCNCPoint4[22195] = {X 274.8846, Y 18.1954, Z -6.3333, A 0.000, B 0.000, C 0.000 }
gfCNCPoint4[22196] = {X 274.8845, Y 38.9911, Z -6.3333, A 0.000, B 0.000, C 0.000 }
gfCNCPoint4[22197] = {X 275.3140, Y 39.7328, Z -6.3333, A 0.000, B 0.000, C 0.000 }
gfCNCPoint4[22198] = {X 275.6763, Y 40.5096, Z -6.3333, A 0.000, B 0.000, C 0.000 }
gfCNCPoint4[22199] = {X 276.0372, Y 39.7353, Z -6.3333, A 0.000, B 0.000, C 0.000 }
gfCNCPoint4[22200] = {X 276.4647, Y 38.9957, Z -6.3333, A 0.000, B 0.000, C 0.000 }
gfCNCPoint4[22201] = {X 276.4643, Y 18.1958, Z -6.3333, A 0.000, B 0.000, C 0.000 }
gfCNCPoint4[22202] = {X 276.0359, Y 17.4564, Z -6.3333, A 0.000, B 0.000, C 0.000 }
gfCNCPoint4[22203] = {X 275.6743, Y 16.6820, Z -6.3333, A 0.000, B 0.000, C 0.000 }
gfCNCPoint4[22204] = {X 273.4570, Y 15.7637, Z -6.3333, A 0.000, B 0.000, C 0.000 }
gfCNCPoint4[22205] = {X 273.0267, Y 16.6335, Z -6.3333, A 0.000, B 0.000, C 0.000 }
gfCNCPoint4[22206] = {X 272.4846, Y 17.4383, Z -6.3333, A 0.000, B 0.000, C 0.000 }
gfCNCPoint4[22207] = {X 272.4845, Y 39.7483, Z -6.3333, A 0.000, B 0.000, C 0.000 }
gfCNCPoint4[22208] = {X 273.0277, Y 40.5549, Z -6.3333, A 0.000, B 0.000, C 0.000 }
gfCNCPoint4[22209] = {X 273.4585, Y 41.4268, Z -6.3333, A 0.000, B 0.000, C 0.000 }
gfCNCPoint4[22210] = {X 273.7588, Y 42.3090, Z -6.3333, A 0.000, B 0.000, C 0.000 }
gfCNCPoint4[22211] = {X 273.9439, Y 43.2223, Z -6.3333, A 0.000, B 0.000, C 0.000 }
gfCNCPoint4[22212] = {X 274.0108, Y 44.1519, Z -6.3333, A 0.000, B 0.000, C 0.000 }
gfCNCPoint4[22213] = {X 274.0110, Y 45.0000, Z -6.3333, A 0.000, B 0.000, C 0.000 }
gfCNCPoint4[22214] = {X 273.9884, Y 45.5734, Z -6.3333, A 0.000, B 0.000, C 0.000 }
gfCNCPoint4[22215] = {X 273.9207, Y 46.1433, Z -6.3333, A 0.000, B 0.000, C 0.000 }
gfCNCPoint4[22216] = {X 275.0713, Y 45.9760, Z -6.3333, A 0.000, B 0.000, C 0.000 }
gfCNCPoint4[22217] = {X 276.2327, Y 45.9200, Z -6.3333, A 0.000, B 0.000, C 0.000 }
gfCNCPoint4[22218] = {X 277.3960, Y 45.9200, Z -6.3333, A 0.000, B 0.000, C 0.000 }
gfCNCPoint4[22219] = {X 277.3539, Y 45.4857, Z -6.3333, A 0.000, B 0.000, C 0.000 }
gfCNCPoint4[22220] = {X 277.3378, Y 45.0498, Z -6.3333, A 0.000, B 0.000, C 0.000 }
gfCNCPoint4[22221] = {X 277.3377, Y 44.1994, Z -6.3333, A 0.000, B 0.000, C 0.000 }
gfCNCPoint4[22222] = {X 277.4026, Y 43.2538, Z -6.3333, A 0.000, B 0.000, C 0.000 }
gfCNCPoint4[22223] = {X 277.5891, Y 42.3245, Z -6.3333, A 0.000, B 0.000, C 0.000 }
gfCNCPoint4[22224] = {X 277.8940, Y 41.4271, Z -6.3333, A 0.000, B 0.000, C 0.000 }
gfCNCPoint4[22225] = {X 278.3237, Y 40.5567, Z -6.3333, A 0.000, B 0.000, C 0.000 }
gfCNCPoint4[22226] = {X 278.8647, Y 39.7507, Z -6.3333, A 0.000, B 0.000, C 0.000 }
gfCNCPoint4[22227] = {X 278.8643, Y 17.4387, Z -6.3333, A 0.000, B 0.000, C 0.000 }
gfCNCPoint4[22228] = {X 278.3221, Y 16.6337, Z -6.3333, A 0.000, B 0.000, C 0.000 }
gfCNCPoint4[22229] = {X 277.8917, Y 15.7637, Z -6.3333, A 0.000, B 0.000, C 0.000 }
gfCNCPoint4[22230] = {X 277.5902, Y 14.8788, Z -6.3333, A 0.000, B 0.000, C 0.000 }
gfCNCPoint4[22231] = {X 277.4046, Y 13.9627, Z -6.3333, A 0.000, B 0.000, C 0.000 }
gfCNCPoint4[22232] = {X 277.3379, Y 13.0303, Z -6.3333, A 0.000, B 0.000, C 0.000 }
gfCNCPoint4[22233] = {X 277.3377, Y 12.1868, Z -6.3333, A 0.000, B 0.000, C 0.000 }
gfCNCPoint4[22234] = {X 277.3952, Y 11.2737, Z -6.3333, A 0.000, B 0.000, C 0.000 }
gfCNCPoint4[22235] = {X 277.5667, Y 10.3750, Z -6.3333, A 0.000, B 0.000, C 0.000 }
gfCNCPoint4[22236] = {X 277.8497, Y 9.5049, Z -6.3333, A 0.000, B 0.000, C 0.000 }
gfCNCPoint4[22237] = {X 273.4971, Y 9.5049, Z -6.3333, A 0.000, B 0.000, C 0.000 }
gfCNCPoint4[22238] = {X 273.7803, Y 10.3735, Z -6.3333, A 0.000, B 0.000, C 0.000 }
gfCNCPoint4[22239] = {X 273.9525, Y 11.2707, Z -6.3333, A 0.000, B 0.000, C 0.000 }
gfCNCPoint4[22240] = {X 274.0110, Y 12.1825, Z -6.3333, A 0.000, B 0.000, C 0.000 }
gfCNCPoint4[22241] = {X 274.0107, Y 13.0462, Z -6.3333, A 0.000, B 0.000, C 0.000 }
gfCNCPoint4[22242] = {X 273.9427, Y 13.9732, Z -6.3333, A 0.000, B 0.000, C 0.000 }
gfCNCPoint4[22243] = {X 273.7571, Y 14.8840, Z -6.3333, A 0.000, B 0.000, C 0.000 }
gfCNCPoint4[22244] = {X 273.4570, Y 15.7637, Z -6.3333, A 0.000, B 0.000, C 0.000 }
gfCNCPoint4[22245] = {X 271.2396, Y 14.8453, Z -6.3333, A 0.000, B 0.000, C 0.000 }
gfCNCPoint4[22246] = {X 270.7507, Y 15.7452, Z -6.3333, A 0.000, B 0.000, C 0.000 }
gfCNCPoint4[22247] = {X 270.0846, Y 16.5231, Z -6.3333, A 0.000, B 0.000, C 0.000 }
gfCNCPoint4[22248] = {X 270.0845, Y 40.6635, Z -6.3333, A 0.000, B 0.000, C 0.000 }
gfCNCPoint4[22249] = {X 270.7247, Y 41.4043, Z -6.3333, A 0.000, B 0.000, C 0.000 }
gfCNCPoint4[22250] = {X 271.2041, Y 42.2580, Z -6.3333, A 0.000, B 0.000, C 0.000 }
gfCNCPoint4[22251] = {X 271.5035, Y 43.1901, Z -6.3333, A 0.000, B 0.000, C 0.000 }
gfCNCPoint4[22252] = {X 271.6108, Y 44.1633, Z -6.3333, A 0.000, B 0.000, C 0.000 }
gfCNCPoint4[22253] = {X 271.6110, Y 45.0000, Z -6.3333, A 0.000, B 0.000, C 0.000 }
gfCNCPoint4[22254] = {X 271.5959, Y 45.3844, Z -6.3333, A 0.000, B 0.000, C 0.000 }
gfCNCPoint4[22255] = {X 271.5505, Y 45.7664, Z -6.3333, A 0.000, B 0.000, C 0.000 }
gfCNCPoint4[22256] = {X 271.2989, Y 46.7171, Z -6.3333, A 0.000, B 0.000, C 0.000 }
gfCNCPoint4[22257] = {X 270.8619, Y 47.5982, Z -6.3333, A 0.000, B 0.000, C 0.000 }
gfCNCPoint4[22258] = {X 270.2571, Y 48.3736, Z -6.3333, A 0.000, B 0.000, C 0.000 }
gfCNCPoint4[22259] = {X 269.5090, Y 49.0121, Z -6.3333, A 0.000, B 0.000, C 0.000 }
gfCNCPoint4[22260] = {X 268.6482, Y 49.4876, Z -6.3333, A 0.000, B 0.000, C 0.000 }
gfCNCPoint4[22261] = {X 267.7095, Y 49.7809, Z -6.3333, A 0.000, B 0.000, C 0.000 }
gfCNCPoint4[22262] = {X 266.7310, Y 49.8800, Z -6.3333, A 0.000, B 0.000, C 0.000 }
gfCNCPoint4[22263] = {X 260.2876, Y 49.8800, Z -6.3333, A 0.000, B 0.000, C 0.000 }
gfCNCPoint4[22264] = {X 259.2646, Y 49.7716, Z -6.3333, A 0.000, B 0.000, C 0.000 }
gfCNCPoint4[22265] = {X 258.2870, Y 49.4511, Z -6.3333, A 0.000, B 0.000, C 0.000 }
gfCNCPoint4[22266] = {X 257.3984, Y 48.9328, Z -6.3333, A 0.000, B 0.000, C 0.000 }
gfCNCPoint4[22267] = {X 256.6382, Y 48.2398, Z -6.3333, A 0.000, B 0.000, C 0.000 }
gfCNCPoint4[22268] = {X 256.0401, Y 47.4028, Z -6.3333, A 0.000, B 0.000, C 0.000 }
gfCNCPoint4[22269] = {X 255.6308, Y 46.4590, Z -6.3333, A 0.000, B 0.000, C 0.000 }
gfCNCPoint4[22270] = {X 255.4666, Y 45.7568, Z -6.3333, A 0.000, B 0.000, C 0.000 }
gfCNCPoint4[22271] = {X 255.4077, Y 45.0380, Z -6.3333, A 0.000, B 0.000, C 0.000 }
gfCNCPoint4[22272] = {X 255.4080, Y 44.1416, Z -6.3333, A 0.000, B 0.000, C 0.000 }
gfCNCPoint4[22273] = {X 255.5183, Y 43.1751, Z -6.3333, A 0.000, B 0.000, C 0.000 }
gfCNCPoint4[22274] = {X 255.8181, Y 42.2496, Z -6.3333, A 0.000, B 0.000, C 0.000 }
gfCNCPoint4[22275] = {X 256.2955, Y 41.4020, Z -6.3333, A 0.000, B 0.000, C 0.000 }
gfCNCPoint4[22276] = {X 256.9315, Y 40.6660, Z -6.3333, A 0.000, B 0.000, C 0.000 }
gfCNCPoint4[22277] = {X 256.9315, Y 35.0338, Z -6.3333, A 0.000, B 0.000, C 0.000 }
gfCNCPoint4[22278] = {X 255.1103, Y 35.0338, Z -6.3333, A 0.000, B 0.000, C 0.000 }
gfCNCPoint4[22279] = {X 251.0867, Y 42.8712, Z -6.3333, A 0.000, B 0.000, C 0.000 }
gfCNCPoint4[22280] = {X 251.2237, Y 43.5131, Z -6.3333, A 0.000, B 0.000, C 0.000 }
gfCNCPoint4[22281] = {X 251.2734, Y 44.1675, Z -6.3333, A 0.000, B 0.000, C 0.000 }
gfCNCPoint4[22282] = {X 251.2736, Y 45.0000, Z -6.3333, A 0.000, B 0.000, C 0.000 }
gfCNCPoint4[22283] = {X 251.2174, Y 45.7380, Z -6.3333, A 0.000, B 0.000, C 0.000 }
gfCNCPoint4[22284] = {X 251.0503, Y 46.4590, Z -6.3333, A 0.000, B 0.000, C 0.000 }
gfCNCPoint4[22285] = {X 250.6346, Y 47.4142, Z -6.3333, A 0.000, B 0.000, C 0.000 }
gfCNCPoint4[22286] = {X 250.0255, Y 48.2593, Z -6.3333, A 0.000, B 0.000, C 0.000 }
gfCNCPoint4[22287] = {X 249.2510, Y 48.9560, Z -6.3333, A 0.000, B 0.000, C 0.000 }
gfCNCPoint4[22288] = {X 248.3462, Y 49.4723, Z -6.3333, A 0.000, B 0.000, C 0.000 }
gfCNCPoint4[22289] = {X 247.3525, Y 49.7849, Z -6.3333, A 0.000, B 0.000, C 0.000 }
gfCNCPoint4[22290] = {X 246.8754, Y 49.8562, Z -6.3333, A 0.000, B 0.000, C 0.000 }
gfCNCPoint4[22291] = {X 246.3936, Y 49.8800, Z -6.3333, A 0.000, B 0.000, C 0.000 }
gfCNCPoint4[22292] = {X 242.5312, Y 49.8800, Z -6.3333, A 0.000, B 0.000, C 0.000 }
gfCNCPoint4[22293] = {X 242.5312, Y 49.4000, Z -6.3333, A 0.000, B 0.000, C 0.000 }
gfCNCPoint4[22294] = {X 239.8075, Y 49.4000, Z -6.3333, A 0.000, B 0.000, C 0.000 }
gfCNCPoint4[22295] = {X 238.8284, Y 49.2897, Z -6.3333, A 0.000, B 0.000, C 0.000 }
gfCNCPoint4[22296] = {X 237.8984, Y 48.9643, Z -6.3333, A 0.000, B 0.000, C 0.000 }
gfCNCPoint4[22297] = {X 237.0641, Y 48.4401, Z -6.3333, A 0.000, B 0.000, C 0.000 }
gfCNCPoint4[22298] = {X 236.3674, Y 47.7434, Z -6.3333, A 0.000, B 0.000, C 0.000 }
gfCNCPoint4[22299] = {X 235.8432, Y 46.9091, Z -6.3333, A 0.000, B 0.000, C 0.000 }
gfCNCPoint4[22300] = {X 235.5178, Y 45.9791, Z -6.3333, A 0.000, B 0.000, C 0.000 }
gfCNCPoint4[22301] = {X 235.4075, Y 45.0000, Z -6.3333, A 0.000, B 0.000, C 0.000 }
gfCNCPoint4[22302] = {X 235.4079, Y 44.1483, Z -6.3333, A 0.000, B 0.000, C 0.000 }
gfCNCPoint4[22303] = {X 235.5063, Y 43.2816, Z -6.3333, A 0.000, B 0.000, C 0.000 }
gfCNCPoint4[22304] = {X 235.7737, Y 42.4514, Z -6.3333, A 0.000, B 0.000, C 0.000 }
gfCNCPoint4[22305] = {X 236.1996, Y 41.6903, Z -6.3333, A 0.000, B 0.000, C 0.000 }
gfCNCPoint4[22306] = {X 236.7672, Y 41.0281, Z -6.3333, A 0.000, B 0.000, C 0.000 }
gfCNCPoint4[22307] = {X 237.4544, Y 40.4909, Z -6.3333, A 0.000, B 0.000, C 0.000 }
gfCNCPoint4[22308] = {X 238.2339, Y 40.0998, Z -6.3333, A 0.000, B 0.000, C 0.000 }
gfCNCPoint4[22309] = {X 242.1745, Y 32.3865, Z -6.3333, A 0.000, B 0.000, C 0.000 }
gfCNCPoint4[22310] = {X 241.0109, Y 31.5940, Z -6.3333, A 0.000, B 0.000, C 0.000 }
gfCNCPoint4[22311] = {X 239.9539, Y 30.6641, Z -6.3333, A 0.000, B 0.000, C 0.000 }
gfCNCPoint4[22312] = {X 239.0195, Y 29.6110, Z -6.3333, A 0.000, B 0.000, C 0.000 }
gfCNCPoint4[22313] = {X 238.2220, Y 28.4507, Z -6.3333, A 0.000, B 0.000, C 0.000 }
gfCNCPoint4[22314] = {X 237.5737, Y 27.2010, Z -6.3333, A 0.000, B 0.000, C 0.000 }
gfCNCPoint4[22315] = {X 237.0843, Y 25.8809, Z -6.3333, A 0.000, B 0.000, C 0.000 }
gfCNCPoint4[22316] = {X 236.6625, Y 24.0613, Z -6.3333, A 0.000, B 0.000, C 0.000 }
gfCNCPoint4[22317] = {X 236.4477, Y 22.2057, Z -6.3333, A 0.000, B 0.000, C 0.000 }
gfCNCPoint4[22318] = {X 236.4425, Y 20.3378, Z -6.3333, A 0.000, B 0.000, C 0.000 }
gfCNCPoint4[22319] = {X 236.6469, Y 18.4811, Z -6.3333, A 0.000, B 0.000, C 0.000 }
gfCNCPoint4[22320] = {X 237.0585, Y 16.6591, Z -6.3333, A 0.000, B 0.000, C 0.000 }
gfCNCPoint4[22321] = {X 237.6328, Y 15.0727, Z -6.3333, A 0.000, B 0.000, C 0.000 }
gfCNCPoint4[22322] = {X 238.4252, Y 13.5833, Z -6.3333, A 0.000, B 0.000, C 0.000 }
gfCNCPoint4[22323] = {X 239.4197, Y 12.2205, Z -6.3333, A 0.000, B 0.000, C 0.000 }
gfCNCPoint4[22324] = {X 240.5966, Y 11.0116, Z -6.3333, A 0.000, B 0.000, C 0.000 }
gfCNCPoint4[22325] = {X 241.9322, Y 9.9808, Z -6.3333, A 0.000, B 0.000, C 0.000 }
gfCNCPoint4[22326] = {X 243.3998, Y 9.1487, Z -6.3333, A 0.000, B 0.000, C 0.000 }
gfCNCPoint4[22327] = {X 244.9702, Y 8.5320, Z -6.3333, A 0.000, B 0.000, C 0.000 }
gfCNCPoint4[22328] = {X 246.6119, Y 8.1430, Z -6.3333, A 0.000, B 0.000, C 0.000 }
gfCNCPoint4[22329] = {X 248.7155, Y 7.8707, Z -6.3333, A 0.000, B 0.000, C 0.000 }
gfCNCPoint4[22330] = {X 250.8352, Y 7.7899, Z -6.3333, A 0.000, B 0.000, C 0.000 }
gfCNCPoint4[22331] = {X 266.7640, Y 7.7899, Z -6.3333, A 0.000, B 0.000, C 0.000 }
gfCNCPoint4[22332] = {X 267.7370, Y 7.9068, Z -6.3333, A 0.000, B 0.000, C 0.000 }
gfCNCPoint4[22333] = {X 268.6600, Y 8.2360, Z -6.3333, A 0.000, B 0.000, C 0.000 }
gfCNCPoint4[22334] = {X 269.4873, Y 8.7613, Z -6.3333, A 0.000, B 0.000, C 0.000 }
gfCNCPoint4[22335] = {X 270.1779, Y 9.4566, Z -6.3333, A 0.000, B 0.000, C 0.000 }
gfCNCPoint4[22336] = {X 270.6976, Y 10.2874, Z -6.3333, A 0.000, B 0.000, C 0.000 }
gfCNCPoint4[22337] = {X 271.0207, Y 11.2126, Z -6.3333, A 0.000, B 0.000, C 0.000 }
gfCNCPoint4[22338] = {X 271.1310, Y 12.1863, Z -6.3333, A 0.000, B 0.000, C 0.000 }
gfCNCPoint4[22339] = {X 271.1308, Y 13.0233, Z -6.3333, A 0.000, B 0.000, C 0.000 }
gfCNCPoint4[22340] = {X 271.0226, Y 13.9490, Z -6.3333, A 0.000, B 0.000, C 0.000 }
gfCNCPoint4[22341] = {X 270.7218, Y 14.8311, Z -6.3333, A 0.000, B 0.000, C 0.000 }
gfCNCPoint4[22342] = {X 270.2420, Y 15.6301, Z -6.3333, A 0.000, B 0.000, C 0.000 }
gfCNCPoint4[22343] = {X 269.6046, Y 16.3100, Z -6.3333, A 0.000, B 0.000, C 0.000 }
gfCNCPoint4[22344] = {X 269.6045, Y 40.8766, Z -6.3333, A 0.000, B 0.000, C 0.000 }
gfCNCPoint4[22345] = {X 270.2487, Y 41.5657, Z -6.3333, A 0.000, B 0.000, C 0.000 }
gfCNCPoint4[22346] = {X 270.7312, Y 42.3762, Z -6.3333, A 0.000, B 0.000, C 0.000 }
gfCNCPoint4[22347] = {X 271.0299, Y 43.2710, Z -6.3333, A 0.000, B 0.000, C 0.000 }
gfCNCPoint4[22348] = {X 271.1310, Y 44.2089, Z -6.3333, A 0.000, B 0.000, C 0.000 }
gfCNCPoint4[22349] = {X 271.1310, Y 45.0000, Z -6.3333, A 0.000, B 0.000, C 0.000 }
gfCNCPoint4[22350] = {X 271.0207, Y 45.9791, Z -6.3333, A 0.000, B 0.000, C 0.000 }
gfCNCPoint4[22351] = {X 270.6953, Y 46.9091, Z -6.3333, A 0.000, B 0.000, C 0.000 }
gfCNCPoint4[22352] = {X 270.1711, Y 47.7434, Z -6.3333, A 0.000, B 0.000, C 0.000 }
gfCNCPoint4[22353] = {X 269.4744, Y 48.4401, Z -6.3333, A 0.000, B 0.000, C 0.000 }
gfCNCPoint4[22354] = {X 268.6401, Y 48.9643, Z -6.3333, A 0.000, B 0.000, C 0.000 }
gfCNCPoint4[22355] = {X 267.7101, Y 49.2897, Z -6.3333, A 0.000, B 0.000, C 0.000 }
gfCNCPoint4[22356] = {X 266.7310, Y 49.4000, Z -6.3333, A 0.000, B 0.000, C 0.000 }
gfCNCPoint4[22357] = {X 260.2876, Y 49.4000, Z -6.3333, A 0.000, B 0.000, C 0.000 }
gfCNCPoint4[22358] = {X 259.3085, Y 49.2897, Z -6.3333, A 0.000, B 0.000, C 0.000 }
gfCNCPoint4[22359] = {X 258.3785, Y 48.9643, Z -6.3333, A 0.000, B 0.000, C 0.000 }
gfCNCPoint4[22360] = {X 257.5442, Y 48.4401, Z -6.3333, A 0.000, B 0.000, C 0.000 }
gfCNCPoint4[22361] = {X 256.8475, Y 47.7433, Z -6.3333, A 0.000, B 0.000, C 0.000 }
gfCNCPoint4[22362] = {X 256.3233, Y 46.9091, Z -6.3333, A 0.000, B 0.000, C 0.000 }
gfCNCPoint4[22363] = {X 255.9979, Y 45.9791, Z -6.3333, A 0.000, B 0.000, C 0.000 }
gfCNCPoint4[22364] = {X 255.8876, Y 45.0000, Z -6.3333, A 0.000, B 0.000, C 0.000 }
gfCNCPoint4[22365] = {X 255.8880, Y 44.1483, Z -6.3333, A 0.000, B 0.000, C 0.000 }
gfCNCPoint4[22366] = {X 255.9984, Y 43.2275, Z -6.3333, A 0.000, B 0.000, C 0.000 }
gfCNCPoint4[22367] = {X 256.2993, Y 42.3503, Z -6.3333, A 0.000, B 0.000, C 0.000 }
gfCNCPoint4[22368] = {X 256.7775, Y 41.5556, Z -6.3333, A 0.000, B 0.000, C 0.000 }
gfCNCPoint4[22369] = {X 257.4115, Y 40.8789, Z -6.3333, A 0.000, B 0.000, C 0.000 }
gfCNCPoint4[22370] = {X 257.4115, Y 34.5538, Z -6.3333, A 0.000, B 0.000, C 0.000 }
gfCNCPoint4[22371] = {X 254.8172, Y 34.5538, Z -6.3333, A 0.000, B 0.000, C 0.000 }
gfCNCPoint4[22372] = {X 250.5705, Y 42.8256, Z -6.3333, A 0.000, B 0.000, C 0.000 }
gfCNCPoint4[22373] = {X 250.7374, Y 43.5083, Z -6.3333, A 0.000, B 0.000, C 0.000 }
gfCNCPoint4[22374] = {X 250.7936, Y 44.2089, Z -6.3333, A 0.000, B 0.000, C 0.000 }
gfCNCPoint4[22375] = {X 250.7936, Y 45.0000, Z -6.3333, A 0.000, B 0.000, C 0.000 }
gfCNCPoint4[22376] = {X 250.6832, Y 45.9791, Z -6.3333, A 0.000, B 0.000, C 0.000 }
gfCNCPoint4[22377] = {X 250.3578, Y 46.9091, Z -6.3333, A 0.000, B 0.000, C 0.000 }
gfCNCPoint4[22378] = {X 249.8336, Y 47.7434, Z -6.3333, A 0.000, B 0.000, C 0.000 }
gfCNCPoint4[22379] = {X 249.1369, Y 48.4401, Z -6.3333, A 0.000, B 0.000, C 0.000 }
gfCNCPoint4[22380] = {X 248.3026, Y 48.9643, Z -6.3333, A 0.000, B 0.000, C 0.000 }
gfCNCPoint4[22381] = {X 247.3727, Y 49.2897, Z -6.3333, A 0.000, B 0.000, C 0.000 }
gfCNCPoint4[22382] = {X 246.3936, Y 49.4000, Z -6.3333, A 0.000, B 0.000, C 0.000 }
gfCNCPoint4[22383] = {X 242.5312, Y 49.4000, Z -6.3333, A 0.000, B 0.000, C 0.000 }
gfCNCPoint4[22384] = {X 242.5312, Y 49.8800, Z -6.3333, A 0.000, B 0.000, C 0.000 }
gfCNCPoint4[22385] = {X 243.4812, Y 50.5824, Z -6.3333, A 0.000, B 0.000, C 0.000 }
gfCNCPoint4[22386] = {X 244.3384, Y 51.3953, Z -6.3333, A 0.000, B 0.000, C 0.000 }
gfCNCPoint4[22387] = {X 245.0903, Y 52.3066, Z -6.3333, A 0.000, B 0.000, C 0.000 }
gfCNCPoint4[22388] = {X 245.7256, Y 53.3027, Z -6.3333, A 0.000, B 0.000, C 0.000 }
gfCNCPoint4[22389] = {X 245.9754, Y 53.7842, Z -6.3333, A 0.000, B 0.000, C 0.000 }
gfCNCPoint4[22390] = {X 246.1979, Y 54.2789, Z -6.3333, A 0.000, B 0.000, C 0.000 }
gfCNCPoint4[22391] = {X 250.0859, Y 55.7950, Z -6.3333, A 0.000, B 0.000, C 0.000 }
gfCNCPoint4[22392] = {X 251.8782, Y 56.5064, Z -6.3333, A 0.000, B 0.000, C 0.000 }
gfCNCPoint4[22393] = {X 253.6490, Y 52.0450, Z -6.3333, A 0.000, B 0.000, C 0.000 }
gfCNCPoint4[22394] = {X 253.4931, Y 51.8947, Z -6.3333, A 0.000, B 0.000, C 0.000 }
gfCNCPoint4[22395] = {X 253.3406, Y 51.7410, Z -6.3333, A 0.000, B 0.000, C 0.000 }
gfCNCPoint4[22396] = {X 253.2764, Y 51.8065, Z -6.3333, A 0.000, B 0.000, C 0.000 }
gfCNCPoint4[22397] = {X 253.2116, Y 51.8714, Z -6.3333, A 0.000, B 0.000, C 0.000 }
gfCNCPoint4[22398] = {X 253.6490, Y 52.0450, Z -6.3333, A 0.000, B 0.000, C 0.000 }
gfCNCPoint4[22399] = {X 252.7636, Y 54.2757, Z -6.3333, A 0.000, B 0.000, C 0.000 }
gfCNCPoint4[22400] = {X 259.4023, Y 56.9107, Z -6.3333, A 0.000, B 0.000, C 0.000 }
gfCNCPoint4[22401] = {X 260.2877, Y 54.6800, Z -6.3333, A 0.000, B 0.000, C 0.000 }
gfCNCPoint4[22402] = {X 261.9958, Y 55.3580, Z -6.3333, A 0.000, B 0.000, C 0.000 }
gfCNCPoint4[22403] = {X 262.0630, Y 55.0181, Z -6.3333, A 0.000, B 0.000, C 0.000 }
gfCNCPoint4[22404] = {X 262.1384, Y 54.6800, Z -6.3333, A 0.000, B 0.000, C 0.000 }
gfCNCPoint4[22405] = {X 260.2877, Y 54.6800, Z -6.3333, A 0.000, B 0.000, C 0.000 }
gfCNCPoint4[22406] = {X 259.4023, Y 56.9107, Z -6.3333, A 0.000, B 0.000, C 0.000 }
gfCNCPoint4[22407] = {X 264.1528, Y 58.7963, Z -6.3333, A 0.000, B 0.000, C 0.000 }
gfCNCPoint4[22408] = {X 264.1527, Y 58.0000, Z -6.3333, A 0.000, B 0.000, C 0.000 }
gfCNCPoint4[22409] = {X 264.2035, Y 56.8933, Z -6.3333, A 0.000, B 0.000, C 0.000 }
gfCNCPoint4[22410] = {X 264.3555, Y 55.7959, Z -6.3333, A 0.000, B 0.000, C 0.000 }
gfCNCPoint4[22411] = {X 264.4116, Y 55.5124, Z -6.3333, A 0.000, B 0.000, C 0.000 }
gfCNCPoint4[22412] = {X 264.4745, Y 55.2303, Z -6.3333, A 0.000, B 0.000, C 0.000 }
gfCNCPoint4[22413] = {X 264.9369, Y 53.7185, Z -6.3333, A 0.000, B 0.000, C 0.000 }
gfCNCPoint4[22414] = {X 265.5928, Y 52.2800, Z -6.3333, A 0.000, B 0.000, C 0.000 }
gfCNCPoint4[22415] = {X 260.2876, Y 52.2800, Z -6.3333, A 0.000, B 0.000, C 0.000 }
gfCNCPoint4[22416] = {X 259.1914, Y 52.1970, Z -6.3333, A 0.000, B 0.000, C 0.000 }
gfCNCPoint4[22417] = {X 258.1203, Y 51.9499, Z -6.3333, A 0.000, B 0.000, C 0.000 }
gfCNCPoint4[22418] = {X 257.0986, Y 51.5444, Z -6.3333, A 0.000, B 0.000, C 0.000 }
gfCNCPoint4[22419] = {X 256.1496, Y 50.9896, Z -6.3333, A 0.000, B 0.000, C 0.000 }
gfCNCPoint4[22420] = {X 255.2949, Y 50.2983, Z -6.3333, A 0.000, B 0.000, C 0.000 }
gfCNCPoint4[22421] = {X 255.1777, Y 50.1853, Z -6.3333, A 0.000, B 0.000, C 0.000 }
gfCNCPoint4[22422] = {X 255.0630, Y 50.0697, Z -6.3333, A 0.000, B 0.000, C 0.000 }
gfCNCPoint4[22423] = {X 254.3405, Y 49.1989, Z -6.3333, A 0.000, B 0.000, C 0.000 }
gfCNCPoint4[22424] = {X 253.7617, Y 48.2267, Z -6.3333, A 0.000, B 0.000, C 0.000 }
gfCNCPoint4[22425] = {X 253.3406, Y 47.1766, Z -6.3333, A 0.000, B 0.000, C 0.000 }
gfCNCPoint4[22426] = {X 252.9194, Y 48.2267, Z -6.3333, A 0.000, B 0.000, C 0.000 }
gfCNCPoint4[22427] = {X 252.3406, Y 49.1989, Z -6.3333, A 0.000, B 0.000, C 0.000 }
gfCNCPoint4[22428] = {X 251.6182, Y 50.0697, Z -6.3333, A 0.000, B 0.000, C 0.000 }
gfCNCPoint4[22429] = {X 251.5699, Y 50.1190, Z -6.3333, A 0.000, B 0.000, C 0.000 }
gfCNCPoint4[22430] = {X 251.5212, Y 50.1677, Z -6.3333, A 0.000, B 0.000, C 0.000 }
gfCNCPoint4[22431] = {X 250.7153, Y 50.8584, Z -6.3333, A 0.000, B 0.000, C 0.000 }
gfCNCPoint4[22432] = {X 249.8174, Y 51.4246, Z -6.3333, A 0.000, B 0.000, C 0.000 }
gfCNCPoint4[22433] = {X 248.8468, Y 51.8542, Z -6.3333, A 0.000, B 0.000, C 0.000 }
gfCNCPoint4[22434] = {X 247.8241, Y 52.1381, Z -6.3333, A 0.000, B 0.000, C 0.000 }
gfCNCPoint4[22435] = {X 247.8928, Y 52.2636, Z -6.3333, A 0.000, B 0.000, C 0.000 }
gfCNCPoint4[22436] = {X 247.9600, Y 52.3900, Z -6.3333, A 0.000, B 0.000, C 0.000 }
gfCNCPoint4[22437] = {X 250.9678, Y 53.5629, Z -6.3333, A 0.000, B 0.000, C 0.000 }
gfCNCPoint4[22438] = {X 252.7636, Y 54.2757, Z -6.3333, A 0.000, B 0.000, C 0.000 }
gfCNCPoint4[22439] = {X 251.8782, Y 56.5064, Z -6.3333, A 0.000, B 0.000, C 0.000 }
gfCNCPoint4[22440] = {X 267.2821, Y 62.6205, Z -6.3333, A 0.000, B 0.000, C 0.000 }
gfCNCPoint4[22441] = {X 266.8843, Y 61.4459, Z -6.3333, A 0.000, B 0.000, C 0.000 }
gfCNCPoint4[22442] = {X 266.6398, Y 60.2301, Z -6.3333, A 0.000, B 0.000, C 0.000 }
gfCNCPoint4[22443] = {X 266.5529, Y 58.9930, Z -6.3333, A 0.000, B 0.000, C 0.000 }
gfCNCPoint4[22444] = {X 266.5527, Y 58.0000, Z -6.3333, A 0.000, B 0.000, C 0.000 }
gfCNCPoint4[22445] = {X 266.6262, Y 56.8093, Z -6.3333, A 0.000, B 0.000, C 0.000 }
gfCNCPoint4[22446] = {X 266.8456, Y 55.6367, Z -6.3333, A 0.000, B 0.000, C 0.000 }
gfCNCPoint4[22447] = {X 267.2076, Y 54.5000, Z -6.3333, A 0.000, B 0.000, C 0.000 }
gfCNCPoint4[22448] = {X 267.7067, Y 53.4164, Z -6.3333, A 0.000, B 0.000, C 0.000 }
gfCNCPoint4[22449] = {X 268.4728, Y 52.2132, Z -6.3333, A 0.000, B 0.000, C 0.000 }
gfCNCPoint4[22450] = {X 269.4075, Y 51.1357, Z -6.3333, A 0.000, B 0.000, C 0.000 }
gfCNCPoint4[22451] = {X 270.4903, Y 50.2072, Z -6.3333, A 0.000, B 0.000, C 0.000 }
gfCNCPoint4[22452] = {X 271.6979, Y 49.4479, Z -6.3333, A 0.000, B 0.000, C 0.000 }
gfCNCPoint4[22453] = {X 273.0039, Y 48.8744, Z -6.3333, A 0.000, B 0.000, C 0.000 }
gfCNCPoint4[22454] = {X 274.3800, Y 48.4989, Z -6.3333, A 0.000, B 0.000, C 0.000 }
gfCNCPoint4[22455] = {X 275.3020, Y 48.3648, Z -6.3333, A 0.000, B 0.000, C 0.000 }
gfCNCPoint4[22456] = {X 276.2327, Y 48.3200, Z -6.3333, A 0.000, B 0.000, C 0.000 }
gfCNCPoint4[22457] = {X 281.0411, Y 48.3200, Z -6.3333, A 0.000, B 0.000, C 0.000 }
gfCNCPoint4[22458] = {X 280.4347, Y 47.5134, Z -6.3333, A 0.000, B 0.000, C 0.000 }
gfCNCPoint4[22459] = {X 280.0072, Y 46.5992, Z -6.3333, A 0.000, B 0.000, C 0.000 }
gfCNCPoint4[22460] = {X 279.7768, Y 45.6167, Z -6.3333, A 0.000, B 0.000, C 0.000 }
gfCNCPoint4[22461] = {X 279.7488, Y 45.3288, Z -6.3333, A 0.000, B 0.000, C 0.000 }
gfCNCPoint4[22462] = {X 279.7378, Y 45.0398, Z -6.3333, A 0.000, B 0.000, C 0.000 }
gfCNCPoint4[22463] = {X 279.7377, Y 44.2048, Z -6.3333, A 0.000, B 0.000, C 0.000 }
gfCNCPoint4[22464] = {X 279.8416, Y 43.2210, Z -6.3333, A 0.000, B 0.000, C 0.000 }
gfCNCPoint4[22465] = {X 280.1400, Y 42.2777, Z -6.3333, A 0.000, B 0.000, C 0.000 }
gfCNCPoint4[22466] = {X 280.6208, Y 41.4132, Z -6.3333, A 0.000, B 0.000, C 0.000 }
gfCNCPoint4[22467] = {X 281.2647, Y 40.6621, Z -6.3333, A 0.000, B 0.000, C 0.000 }
gfCNCPoint4[22468] = {X 281.2643, Y 16.5233, Z -6.3333, A 0.000, B 0.000, C 0.000 }
gfCNCPoint4[22469] = {X 280.6235, Y 15.7818, Z -6.3333, A 0.000, B 0.000, C 0.000 }
gfCNCPoint4[22470] = {X 280.1438, Y 14.9272, Z -6.3333, A 0.000, B 0.000, C 0.000 }
gfCNCPoint4[22471] = {X 279.8446, Y 13.9940, Z -6.3333, A 0.000, B 0.000, C 0.000 }
gfCNCPoint4[22472] = {X 279.7378, Y 13.0198, Z -6.3333, A 0.000, B 0.000, C 0.000 }
gfCNCPoint4[22473] = {X 279.7377, Y 12.1868, Z -6.3333, A 0.000, B 0.000, C 0.000 }
gfCNCPoint4[22474] = {X 279.8242, Y 11.2717, Z -6.3333, A 0.000, B 0.000, C 0.000 }
gfCNCPoint4[22475] = {X 280.0809, Y 10.3890, Z -6.3333, A 0.000, B 0.000, C 0.000 }
gfCNCPoint4[22476] = {X 280.5256, Y 9.5280, Z -6.3333, A 0.000, B 0.000, C 0.000 }
gfCNCPoint4[22477] = {X 281.1317, Y 8.7718, Z -6.3333, A 0.000, B 0.000, C 0.000 }
gfCNCPoint4[22478] = {X 281.8753, Y 8.1503, Z -6.3333, A 0.000, B 0.000, C 0.000 }
gfCNCPoint4[22479] = {X 282.7270, Y 7.6879, Z -6.3333, A 0.000, B 0.000, C 0.000 }
gfCNCPoint4[22480] = {X 283.6533, Y 7.4030, Z -6.3333, A 0.000, B 0.000, C 0.000 }
gfCNCPoint4[22481] = {X 284.6177, Y 7.3068, Z -6.3333, A 0.000, B 0.000, C 0.000 }
gfCNCPoint4[22482] = {X 291.0611, Y 7.3068, Z -6.3333, A 0.000, B 0.000, C 0.000 }
gfCNCPoint4[22483] = {X 292.0255, Y 7.4030, Z -6.3333, A 0.000, B 0.000, C 0.000 }
gfCNCPoint4[22484] = {X 292.9518, Y 7.6879, Z -6.3333, A 0.000, B 0.000, C 0.000 }
gfCNCPoint4[22485] = {X 293.8035, Y 8.1503, Z -6.3333, A 0.000, B 0.000, C 0.000 }
gfCNCPoint4[22486] = {X 294.5471, Y 8.7718, Z -6.3333, A 0.000, B 0.000, C 0.000 }
gfCNCPoint4[22487] = {X 295.1532, Y 9.5280, Z -6.3333, A 0.000, B 0.000, C 0.000 }
gfCNCPoint4[22488] = {X 295.5979, Y 10.3890, Z -6.3333, A 0.000, B 0.000, C 0.000 }
gfCNCPoint4[22489] = {X 295.8044, Y 11.0396, Z -6.3333, A 0.000, B 0.000, C 0.000 }
gfCNCPoint4[22490] = {X 295.9180, Y 11.7127, Z -6.3333, A 0.000, B 0.000, C 0.000 }
gfCNCPoint4[22491] = {X 295.9354, Y 11.9495, Z -6.3333, A 0.000, B 0.000, C 0.000 }
gfCNCPoint4[22492] = {X 295.9411, Y 12.1868, Z -6.3333, A 0.000, B 0.000, C 0.000 }
gfCNCPoint4[22493] = {X 295.9409, Y 13.0237, Z -6.3333, A 0.000, B 0.000, C 0.000 }
gfCNCPoint4[22494] = {X 295.9342, Y 13.2382, Z -6.3333, A 0.000, B 0.000, C 0.000 }
gfCNCPoint4[22495] = {X 295.9180, Y 13.4521, Z -6.3333, A 0.000, B 0.000, C 0.000 }
gfCNCPoint4[22496] = {X 298.3067, Y 13.6853, Z -6.3333, A 0.000, B 0.000, C 0.000 }
gfCNCPoint4[22497] = {X 298.1362, Y 14.6934, Z -6.3333, A 0.000, B 0.000, C 0.000 }
gfCNCPoint4[22498] = {X 297.8261, Y 15.6676, Z -6.3333, A 0.000, B 0.000, C 0.000 }
gfCNCPoint4[22499] = {X 297.3826, Y 16.5888, Z -6.3333, A 0.000, B 0.000, C 0.000 }
gfCNCPoint4[22500] = {X 296.8144, Y 17.4388, Z -6.3333, A 0.000, B 0.000, C 0.000 }
gfCNCPoint4[22501] = {X 296.8147, Y 19.2365, Z -6.3333, A 0.000, B 0.000, C 0.000 }
gfCNCPoint4[22502] = {X 299.7986, Y 19.2365, Z -6.3333, A 0.000, B 0.000, C 0.000 }
gfCNCPoint4[22503] = {X 299.7987, Y 17.4385, Z -6.3333, A 0.000, B 0.000, C 0.000 }
gfCNCPoint4[22504] = {X 299.2307, Y 16.5885, Z -6.3333, A 0.000, B 0.000, C 0.000 }
gfCNCPoint4[22505] = {X 298.7872, Y 15.6674, Z -6.3333, A 0.000, B 0.000, C 0.000 }
gfCNCPoint4[22506] = {X 298.4772, Y 14.6932, Z -6.3333, A 0.000, B 0.000, C 0.000 }
gfCNCPoint4[22507] = {X 298.3067, Y 13.6853, Z -6.3333, A 0.000, B 0.000, C 0.000 }
gfCNCPoint4[22508] = {X 295.9180, Y 13.4521, Z -6.3333, A 0.000, B 0.000, C 0.000 }
gfCNCPoint4[22509] = {X 295.7560, Y 14.3093, Z -6.3333, A 0.000, B 0.000, C 0.000 }
gfCNCPoint4[22510] = {X 295.4440, Y 15.1239, Z -6.3333, A 0.000, B 0.000, C 0.000 }
gfCNCPoint4[22511] = {X 294.9919, Y 15.8700, Z -6.3333, A 0.000, B 0.000, C 0.000 }
gfCNCPoint4[22512] = {X 294.4142, Y 16.5236, Z -6.3333, A 0.000, B 0.000, C 0.000 }
gfCNCPoint4[22513] = {X 294.4151, Y 21.6365, Z -6.3333, A 0.000, B 0.000, C 0.000 }
gfCNCPoint4[22514] = {X 302.1985, Y 21.6365, Z -6.3333, A 0.000, B 0.000, C 0.000 }
gfCNCPoint4[22515] = {X 302.1988, Y 16.5233, Z -6.3333, A 0.000, B 0.000, C 0.000 }
gfCNCPoint4[22516] = {X 301.6212, Y 15.8697, Z -6.3333, A 0.000, B 0.000, C 0.000 }
gfCNCPoint4[22517] = {X 301.1693, Y 15.1237, Z -6.3333, A 0.000, B 0.000, C 0.000 }
gfCNCPoint4[22518] = {X 300.8573, Y 14.3092, Z -6.3333, A 0.000, B 0.000, C 0.000 }
gfCNCPoint4[22519] = {X 300.6953, Y 13.4521, Z -6.3333, A 0.000, B 0.000, C 0.000 }
gfCNCPoint4[22520] = {X 300.6791, Y 13.2371, Z -6.3333, A 0.000, B 0.000, C 0.000 }
gfCNCPoint4[22521] = {X 300.6724, Y 13.0215, Z -6.3333, A 0.000, B 0.000, C 0.000 }
gfCNCPoint4[22522] = {X 300.6723, Y 12.1868, Z -6.3333, A 0.000, B 0.000, C 0.000 }
gfCNCPoint4[22523] = {X 300.6780, Y 11.9495, Z -6.3333, A 0.000, B 0.000, C 0.000 }
gfCNCPoint4[22524] = {X 300.6953, Y 11.7127, Z -6.3333, A 0.000, B 0.000, C 0.000 }
gfCNCPoint4[22525] = {X 300.8090, Y 11.0396, Z -6.3333, A 0.000, B 0.000, C 0.000 }
gfCNCPoint4[22526] = {X 301.0155, Y 10.3890, Z -6.3333, A 0.000, B 0.000, C 0.000 }
gfCNCPoint4[22527] = {X 301.4602, Y 9.5280, Z -6.3333, A 0.000, B 0.000, C 0.000 }
gfCNCPoint4[22528] = {X 302.0663, Y 8.7718, Z -6.3333, A 0.000, B 0.000, C 0.000 }
gfCNCPoint4[22529] = {X 302.8099, Y 8.1503, Z -6.3333, A 0.000, B 0.000, C 0.000 }
gfCNCPoint4[22530] = {X 303.6616, Y 7.6879, Z -6.3333, A 0.000, B 0.000, C 0.000 }
gfCNCPoint4[22531] = {X 304.5879, Y 7.4030, Z -6.3333, A 0.000, B 0.000, C 0.000 }
gfCNCPoint4[22532] = {X 305.5523, Y 7.3068, Z -6.3333, A 0.000, B 0.000, C 0.000 }
gfCNCPoint4[22533] = {X 311.9957, Y 7.3068, Z -6.3333, A 0.000, B 0.000, C 0.000 }
gfCNCPoint4[22534] = {X 312.9478, Y 7.4006, Z -6.3333, A 0.000, B 0.000, C 0.000 }
gfCNCPoint4[22535] = {X 313.8632, Y 7.6783, Z -6.3333, A 0.000, B 0.000, C 0.000 }
gfCNCPoint4[22536] = {X 314.7069, Y 8.1292, Z -6.3333, A 0.000, B 0.000, C 0.000 }
gfCNCPoint4[22537] = {X 315.4464, Y 8.7361, Z -6.3333, A 0.000, B 0.000, C 0.000 }
gfCNCPoint4[22538] = {X 316.0533, Y 9.4756, Z -6.3333, A 0.000, B 0.000, C 0.000 }
gfCNCPoint4[22539] = {X 316.5043, Y 10.3193, Z -6.3333, A 0.000, B 0.000, C 0.000 }
gfCNCPoint4[22540] = {X 316.7820, Y 11.2348, Z -6.3333, A 0.000, B 0.000, C 0.000 }
gfCNCPoint4[22541] = {X 316.8757, Y 12.1868, Z -6.3333, A 0.000, B 0.000, C 0.000 }
gfCNCPoint4[22542] = {X 316.8755, Y 13.0237, Z -6.3333, A 0.000, B 0.000, C 0.000 }
gfCNCPoint4[22543] = {X 316.7682, Y 13.9967, Z -6.3333, A 0.000, B 0.000, C 0.000 }
gfCNCPoint4[22544] = {X 316.4689, Y 14.9287, Z -6.3333, A 0.000, B 0.000, C 0.000 }
gfCNCPoint4[22545] = {X 315.9895, Y 15.7823, Z -6.3333, A 0.000, B 0.000, C 0.000 }
gfCNCPoint4[22546] = {X 315.3495, Y 16.5229, Z -6.3333, A 0.000, B 0.000, C 0.000 }
gfCNCPoint4[22547] = {X 315.3487, Y 40.6631, Z -6.3333, A 0.000, B 0.000, C 0.000 }
gfCNCPoint4[22548] = {X 315.9895, Y 41.4046, Z -6.3333, A 0.000, B 0.000, C 0.000 }
gfCNCPoint4[22549] = {X 316.4693, Y 42.2591, Z -6.3333, A 0.000, B 0.000, C 0.000 }
gfCNCPoint4[22550] = {X 316.7687, Y 43.1923, Z -6.3333, A 0.000, B 0.000, C 0.000 }
gfCNCPoint4[22551] = {X 316.8755, Y 44.1664, Z -6.3333, A 0.000, B 0.000, C 0.000 }
gfCNCPoint4[22552] = {X 316.8757, Y 45.0000, Z -6.3333, A 0.000, B 0.000, C 0.000 }
gfCNCPoint4[22553] = {X 316.8749, Y 45.0899, Z -6.3333, A 0.000, B 0.000, C 0.000 }
gfCNCPoint4[22554] = {X 316.8724, Y 45.1799, Z -6.3333, A 0.000, B 0.000, C 0.000 }
gfCNCPoint4[22555] = {X 316.8594, Y 45.3987, Z -6.3333, A 0.000, B 0.000, C 0.000 }
gfCNCPoint4[22556] = {X 316.8366, Y 45.6167, Z -6.3333, A 0.000, B 0.000, C 0.000 }
gfCNCPoint4[22557] = {X 316.6062, Y 46.5992, Z -6.3333, A 0.000, B 0.000, C 0.000 }
gfCNCPoint4[22558] = {X 316.1787, Y 47.5134, Z -6.3333, A 0.000, B 0.000, C 0.000 }
gfCNCPoint4[22559] = {X 315.5723, Y 48.3200, Z -6.3333, A 0.000, B 0.000, C 0.000 }
gfCNCPoint4[22560] = {X 315.2205, Y 47.9934, Z -6.3333, A 0.000, B 0.000, C 0.000 }
gfCNCPoint4[22561] = {X 314.5413, Y 48.5889, Z -6.3333, A 0.000, B 0.000, C 0.000 }
gfCNCPoint4[22562] = {X 313.7548, Y 49.0331, Z -6.3333, A 0.000, B 0.000, C 0.000 }
gfCNCPoint4[22563] = {X 312.8942, Y 49.3073, Z -6.3333, A 0.000, B 0.000, C 0.000 }
gfCNCPoint4[22564] = {X 311.9957, Y 49.4000, Z -6.3333, A 0.000, B 0.000, C 0.000 }
gfCNCPoint4[22565] = {X 305.5523, Y 49.4000, Z -6.3333, A 0.000, B 0.000, C 0.000 }
gfCNCPoint4[22566] = {X 304.5732, Y 49.2897, Z -6.3333, A 0.000, B 0.000, C 0.000 }
gfCNCPoint4[22567] = {X 303.6432, Y 48.9643, Z -6.3333, A 0.000, B 0.000, C 0.000 }
gfCNCPoint4[22568] = {X 302.8089, Y 48.4400, Z -6.3333, A 0.000, B 0.000, C 0.000 }
gfCNCPoint4[22569] = {X 302.1122, Y 47.7433, Z -6.3333, A 0.000, B 0.000, C 0.000 }
gfCNCPoint4[22570] = {X 301.5880, Y 46.9091, Z -6.3333, A 0.000, B 0.000, C 0.000 }
gfCNCPoint4[22571] = {X 301.2626, Y 45.9791, Z -6.3333, A 0.000, B 0.000, C 0.000 }
gfCNCPoint4[22572] = {X 301.1523, Y 45.0000, Z -6.3333, A 0.000, B 0.000, C 0.000 }
gfCNCPoint4[22573] = {X 301.1524, Y 44.1995, Z -6.3333, A 0.000, B 0.000, C 0.000 }
gfCNCPoint4[22574] = {X 301.2697, Y 43.2560, Z -6.3333, A 0.000, B 0.000, C 0.000 }
gfCNCPoint4[22575] = {X 301.5725, Y 42.3547, Z -6.3333, A 0.000, B 0.000, C 0.000 }
gfCNCPoint4[22576] = {X 302.0486, Y 41.5318, Z -6.3333, A 0.000, B 0.000, C 0.000 }
gfCNCPoint4[22577] = {X 302.6791, Y 40.8202, Z -6.3333, A 0.000, B 0.000, C 0.000 }
gfCNCPoint4[22578] = {X 302.6791, Y 34.1143, Z -6.3333, A 0.000, B 0.000, C 0.000 }
gfCNCPoint4[22579] = {X 293.9349, Y 34.1143, Z -6.3333, A 0.000, B 0.000, C 0.000 }
gfCNCPoint4[22580] = {X 293.9343, Y 40.8657, Z -6.3333, A 0.000, B 0.000, C 0.000 }
gfCNCPoint4[22581] = {X 294.5743, Y 41.5607, Z -6.3333, A 0.000, B 0.000, C 0.000 }
gfCNCPoint4[22582] = {X 295.0550, Y 42.3741, Z -6.3333, A 0.000, B 0.000, C 0.000 }
gfCNCPoint4[22583] = {X 295.3550, Y 43.2700, Z -6.3333, A 0.000, B 0.000, C 0.000 }
gfCNCPoint4[22584] = {X 295.4611, Y 44.2089, Z -6.3333, A 0.000, B 0.000, C 0.000 }
gfCNCPoint4[22585] = {X 295.4611, Y 45.0000, Z -6.3333, A 0.000, B 0.000, C 0.000 }
gfCNCPoint4[22586] = {X 295.3508, Y 45.9791, Z -6.3333, A 0.000, B 0.000, C 0.000 }
gfCNCPoint4[22587] = {X 295.0254, Y 46.9091, Z -6.3333, A 0.000, B 0.000, C 0.000 }
gfCNCPoint4[22588] = {X 294.5012, Y 47.7434, Z -6.3333, A 0.000, B 0.000, C 0.000 }
gfCNCPoint4[22589] = {X 293.8045, Y 48.4401, Z -6.3333, A 0.000, B 0.000, C 0.000 }
gfCNCPoint4[22590] = {X 292.9702, Y 48.9643, Z -6.3333, A 0.000, B 0.000, C 0.000 }
gfCNCPoint4[22591] = {X 292.0402, Y 49.2897, Z -6.3333, A 0.000, B 0.000, C 0.000 }
gfCNCPoint4[22592] = {X 291.0611, Y 49.4000, Z -6.3333, A 0.000, B 0.000, C 0.000 }
gfCNCPoint4[22593] = {X 284.6177, Y 49.4000, Z -6.3333, A 0.000, B 0.000, C 0.000 }
gfCNCPoint4[22594] = {X 283.6386, Y 49.2897, Z -6.3333, A 0.000, B 0.000, C 0.000 }
gfCNCPoint4[22595] = {X 282.7086, Y 48.9643, Z -6.3333, A 0.000, B 0.000, C 0.000 }
gfCNCPoint4[22596] = {X 281.8743, Y 48.4400, Z -6.3333, A 0.000, B 0.000, C 0.000 }
gfCNCPoint4[22597] = {X 281.1776, Y 47.7433, Z -6.3333, A 0.000, B 0.000, C 0.000 }
gfCNCPoint4[22598] = {X 280.6534, Y 46.9091, Z -6.3333, A 0.000, B 0.000, C 0.000 }
gfCNCPoint4[22599] = {X 280.3280, Y 45.9791, Z -6.3333, A 0.000, B 0.000, C 0.000 }
gfCNCPoint4[22600] = {X 280.2177, Y 45.0000, Z -6.3333, A 0.000, B 0.000, C 0.000 }
gfCNCPoint4[22601] = {X 280.2177, Y 44.2070, Z -6.3333, A 0.000, B 0.000, C 0.000 }
gfCNCPoint4[22602] = {X 280.3220, Y 43.2698, Z -6.3333, A 0.000, B 0.000, C 0.000 }
gfCNCPoint4[22603] = {X 280.6217, Y 42.3758, Z -6.3333, A 0.000, B 0.000, C 0.000 }
gfCNCPoint4[22604] = {X 281.1031, Y 41.5650, Z -6.3333, A 0.000, B 0.000, C 0.000 }
gfCNCPoint4[22605] = {X 281.7447, Y 40.8740, Z -6.3333, A 0.000, B 0.000, C 0.000 }
gfCNCPoint4[22606] = {X 281.7443, Y 16.3103, Z -6.3333, A 0.000, B 0.000, C 0.000 }
gfCNCPoint4[22607] = {X 281.1000, Y 15.6212, Z -6.3333, A 0.000, B 0.000, C 0.000 }
gfCNCPoint4[22608] = {X 280.6175, Y 14.8106, Z -6.3333, A 0.000, B 0.000, C 0.000 }
gfCNCPoint4[22609] = {X 280.3188, Y 13.9159, Z -6.3333, A 0.000, B 0.000, C 0.000 }
gfCNCPoint4[22610] = {X 280.2177, Y 12.9780, Z -6.3333, A 0.000, B 0.000, C 0.000 }
gfCNCPoint4[22611] = {X 280.2177, Y 12.1868, Z -6.3333, A 0.000, B 0.000, C 0.000 }
gfCNCPoint4[22612] = {X 280.3280, Y 11.2077, Z -6.3333, A 0.000, B 0.000, C 0.000 }
gfCNCPoint4[22613] = {X 280.6534, Y 10.2777, Z -6.3333, A 0.000, B 0.000, C 0.000 }
gfCNCPoint4[22614] = {X 281.1776, Y 9.4435, Z -6.3333, A 0.000, B 0.000, C 0.000 }
gfCNCPoint4[22615] = {X 281.8743, Y 8.7468, Z -6.3333, A 0.000, B 0.000, C 0.000 }
gfCNCPoint4[22616] = {X 282.7086, Y 8.2226, Z -6.3333, A 0.000, B 0.000, C 0.000 }
gfCNCPoint4[22617] = {X 283.6386, Y 7.8971, Z -6.3333, A 0.000, B 0.000, C 0.000 }
gfCNCPoint4[22618] = {X 284.6177, Y 7.7868, Z -6.3333, A 0.000, B 0.000, C 0.000 }
gfCNCPoint4[22619] = {X 291.0611, Y 7.7868, Z -6.3333, A 0.000, B 0.000, C 0.000 }
gfCNCPoint4[22620] = {X 292.0402, Y 7.8971, Z -6.3333, A 0.000, B 0.000, C 0.000 }
gfCNCPoint4[22621] = {X 292.9702, Y 8.2226, Z -6.3333, A 0.000, B 0.000, C 0.000 }
gfCNCPoint4[22622] = {X 293.8045, Y 8.7468, Z -6.3333, A 0.000, B 0.000, C 0.000 }
gfCNCPoint4[22623] = {X 294.5012, Y 9.4435, Z -6.3333, A 0.000, B 0.000, C 0.000 }
gfCNCPoint4[22624] = {X 295.0254, Y 10.2777, Z -6.3333, A 0.000, B 0.000, C 0.000 }
gfCNCPoint4[22625] = {X 295.3508, Y 11.2077, Z -6.3333, A 0.000, B 0.000, C 0.000 }
gfCNCPoint4[22626] = {X 295.4611, Y 12.1868, Z -6.3333, A 0.000, B 0.000, C 0.000 }
gfCNCPoint4[22627] = {X 295.4609, Y 13.0233, Z -6.3333, A 0.000, B 0.000, C 0.000 }
gfCNCPoint4[22628] = {X 295.3526, Y 13.9492, Z -6.3333, A 0.000, B 0.000, C 0.000 }
gfCNCPoint4[22629] = {X 295.0517, Y 14.8314, Z -6.3333, A 0.000, B 0.000, C 0.000 }
gfCNCPoint4[22630] = {X 294.5717, Y 15.6305, Z -6.3333, A 0.000, B 0.000, C 0.000 }
gfCNCPoint4[22631] = {X 293.9342, Y 16.3105, Z -6.3333, A 0.000, B 0.000, C 0.000 }
gfCNCPoint4[22632] = {X 293.9352, Y 22.1165, Z -6.3333, A 0.000, B 0.000, C 0.000 }
gfCNCPoint4[22633] = {X 302.6785, Y 22.1165, Z -6.3333, A 0.000, B 0.000, C 0.000 }
gfCNCPoint4[22634] = {X 302.6788, Y 16.3102, Z -6.3333, A 0.000, B 0.000, C 0.000 }
gfCNCPoint4[22635] = {X 302.0346, Y 15.6211, Z -6.3333, A 0.000, B 0.000, C 0.000 }
gfCNCPoint4[22636] = {X 301.5520, Y 14.8106, Z -6.3333, A 0.000, B 0.000, C 0.000 }
gfCNCPoint4[22637] = {X 301.2534, Y 13.9158, Z -6.3333, A 0.000, B 0.000, C 0.000 }
gfCNCPoint4[22638] = {X 301.1523, Y 12.9780, Z -6.3333, A 0.000, B 0.000, C 0.000 }
gfCNCPoint4[22639] = {X 301.1523, Y 12.1868, Z -6.3333, A 0.000, B 0.000, C 0.000 }
gfCNCPoint4[22640] = {X 301.2626, Y 11.2077, Z -6.3333, A 0.000, B 0.000, C 0.000 }
gfCNCPoint4[22641] = {X 301.5880, Y 10.2777, Z -6.3333, A 0.000, B 0.000, C 0.000 }
gfCNCPoint4[22642] = {X 302.1122, Y 9.4435, Z -6.3333, A 0.000, B 0.000, C 0.000 }
gfCNCPoint4[22643] = {X 302.8089, Y 8.7468, Z -6.3333, A 0.000, B 0.000, C 0.000 }
gfCNCPoint4[22644] = {X 303.6432, Y 8.2226, Z -6.3333, A 0.000, B 0.000, C 0.000 }
gfCNCPoint4[22645] = {X 304.5732, Y 7.8971, Z -6.3333, A 0.000, B 0.000, C 0.000 }
gfCNCPoint4[22646] = {X 305.5523, Y 7.7868, Z -6.3333, A 0.000, B 0.000, C 0.000 }
gfCNCPoint4[22647] = {X 311.9957, Y 7.7868, Z -6.3333, A 0.000, B 0.000, C 0.000 }
gfCNCPoint4[22648] = {X 312.9748, Y 7.8971, Z -6.3333, A 0.000, B 0.000, C 0.000 }
gfCNCPoint4[22649] = {X 313.9048, Y 8.2226, Z -6.3333, A 0.000, B 0.000, C 0.000 }
gfCNCPoint4[22650] = {X 314.7391, Y 8.7468, Z -6.3333, A 0.000, B 0.000, C 0.000 }
gfCNCPoint4[22651] = {X 315.4358, Y 9.4435, Z -6.3333, A 0.000, B 0.000, C 0.000 }
gfCNCPoint4[22652] = {X 315.9600, Y 10.2777, Z -6.3333, A 0.000, B 0.000, C 0.000 }
gfCNCPoint4[22653] = {X 316.2854, Y 11.2077, Z -6.3333, A 0.000, B 0.000, C 0.000 }
gfCNCPoint4[22654] = {X 316.3957, Y 12.1868, Z -6.3333, A 0.000, B 0.000, C 0.000 }
gfCNCPoint4[22655] = {X 316.3955, Y 13.0233, Z -6.3333, A 0.000, B 0.000, C 0.000 }
gfCNCPoint4[22656] = {X 316.2873, Y 13.9489, Z -6.3333, A 0.000, B 0.000, C 0.000 }
gfCNCPoint4[22657] = {X 315.9865, Y 14.8310, Z -6.3333, A 0.000, B 0.000, C 0.000 }
gfCNCPoint4[22658] = {X 315.5068, Y 15.6299, Z -6.3333, A 0.000, B 0.000, C 0.000 }
gfCNCPoint4[22659] = {X 314.8695, Y 16.3099, Z -6.3333, A 0.000, B 0.000, C 0.000 }
gfCNCPoint4[22660] = {X 314.8687, Y 40.8762, Z -6.3333, A 0.000, B 0.000, C 0.000 }
gfCNCPoint4[22661] = {X 315.5131, Y 41.5653, Z -6.3333, A 0.000, B 0.000, C 0.000 }
gfCNCPoint4[22662] = {X 315.9958, Y 42.3760, Z -6.3333, A 0.000, B 0.000, C 0.000 }
gfCNCPoint4[22663] = {X 316.2946, Y 43.2709, Z -6.3333, A 0.000, B 0.000, C 0.000 }
gfCNCPoint4[22664] = {X 316.3957, Y 44.2089, Z -6.3333, A 0.000, B 0.000, C 0.000 }
gfCNCPoint4[22665] = {X 316.3957, Y 45.0000, Z -6.3333, A 0.000, B 0.000, C 0.000 }
gfCNCPoint4[22666] = {X 316.3190, Y 45.8182, Z -6.3333, A 0.000, B 0.000, C 0.000 }
gfCNCPoint4[22667] = {X 316.0914, Y 46.6079, Z -6.3333, A 0.000, B 0.000, C 0.000 }
gfCNCPoint4[22668] = {X 315.7209, Y 47.3415, Z -6.3333, A 0.000, B 0.000, C 0.000 }
gfCNCPoint4[22669] = {X 315.2205, Y 47.9934, Z -6.3333, A 0.000, B 0.000, C 0.000 }
gfCNCPoint4[22670] = {X 315.5723, Y 48.3200, Z -6.3333, A 0.000, B 0.000, C 0.000 }
gfCNCPoint4[22671] = {X 324.3107, Y 48.3200, Z -6.3333, A 0.000, B 0.000, C 0.000 }
gfCNCPoint4[22672] = {X 325.5555, Y 48.4004, Z -6.3333, A 0.000, B 0.000, C 0.000 }
gfCNCPoint4[22673] = {X 326.7797, Y 48.6402, Z -6.3333, A 0.000, B 0.000, C 0.000 }
gfCNCPoint4[22674] = {X 325.5882, Y 48.0963, Z -6.3333, A 0.000, B 0.000, C 0.000 }
gfCNCPoint4[22675] = {X 324.4810, Y 47.3966, Z -6.3333, A 0.000, B 0.000, C 0.000 }
gfCNCPoint4[22676] = {X 323.4784, Y 46.5538, Z -6.3333, A 0.000, B 0.000, C 0.000 }
gfCNCPoint4[22677] = {X 322.8382, Y 45.9295, Z -6.3333, A 0.000, B 0.000, C 0.000 }
gfCNCPoint4[22678] = {X 322.2180, Y 45.2650, Z -6.3333, A 0.000, B 0.000, C 0.000 }
gfCNCPoint4[22679] = {X 321.6628, Y 44.5452, Z -6.3333, A 0.000, B 0.000, C 0.000 }
gfCNCPoint4[22680] = {X 323.6300, Y 43.1703, Z -6.3333, A 0.000, B 0.000, C 0.000 }
gfCNCPoint4[22681] = {X 323.0063, Y 42.0918, Z -6.3333, A 0.000, B 0.000, C 0.000 }
gfCNCPoint4[22682] = {X 322.5757, Y 40.9227, Z -6.3333, A 0.000, B 0.000, C 0.000 }
gfCNCPoint4[22683] = {X 322.3506, Y 39.6973, Z -6.3333, A 0.000, B 0.000, C 0.000 }
gfCNCPoint4[22684] = {X 322.3379, Y 38.4514, Z -6.3333, A 0.000, B 0.000, C 0.000 }
gfCNCPoint4[22685] = {X 322.5377, Y 37.2217, Z -6.3333, A 0.000, B 0.000, C 0.000 }
gfCNCPoint4[22686] = {X 322.9443, Y 36.0440, Z -6.3333, A 0.000, B 0.000, C 0.000 }
gfCNCPoint4[22687] = {X 323.5458, Y 34.9529, Z -6.3333, A 0.000, B 0.000, C 0.000 }
gfCNCPoint4[22688] = {X 327.8179, Y 28.5658, Z -6.3333, A 0.000, B 0.000, C 0.000 }
gfCNCPoint4[22689] = {X 328.5476, Y 27.6613, Z -6.3333, A 0.000, B 0.000, C 0.000 }
gfCNCPoint4[22690] = {X 329.4120, Y 26.8845, Z -6.3333, A 0.000, B 0.000, C 0.000 }
gfCNCPoint4[22691] = {X 330.3889, Y 26.2552, Z -6.3333, A 0.000, B 0.000, C 0.000 }
gfCNCPoint4[22692] = {X 331.5063, Y 25.7713, Z -6.3333, A 0.000, B 0.000, C 0.000 }
gfCNCPoint4[22693] = {X 332.6887, Y 25.4804, Z -6.3333, A 0.000, B 0.000, C 0.000 }
gfCNCPoint4[22694] = {X 333.9031, Y 25.3907, Z -6.3333, A 0.000, B 0.000, C 0.000 }
gfCNCPoint4[22695] = {X 335.1154, Y 25.5046, Z -6.3333, A 0.000, B 0.000, C 0.000 }
gfCNCPoint4[22696] = {X 336.2918, Y 25.8191, Z -6.3333, A 0.000, B 0.000, C 0.000 }
gfCNCPoint4[22697] = {X 337.3993, Y 26.3252, Z -6.3333, A 0.000, B 0.000, C 0.000 }
gfCNCPoint4[22698] = {X 338.1753, Y 26.8291, Z -6.3333, A 0.000, B 0.000, C 0.000 }
gfCNCPoint4[22699] = {X 338.8812, Y 27.4274, Z -6.3333, A 0.000, B 0.000, C 0.000 }
gfCNCPoint4[22700] = {X 339.4514, Y 27.9767, Z -6.3333, A 0.000, B 0.000, C 0.000 }
gfCNCPoint4[22701] = {X 339.8232, Y 28.3622, Z -6.3333, A 0.000, B 0.000, C 0.000 }
gfCNCPoint4[22702] = {X 340.1656, Y 28.7740, Z -6.3333, A 0.000, B 0.000, C 0.000 }
gfCNCPoint4[22703] = {X 345.8671, Y 24.3770, Z -6.3333, A 0.000, B 0.000, C 0.000 }
gfCNCPoint4[22704] = {X 346.4655, Y 25.2127, Z -6.3333, A 0.000, B 0.000, C 0.000 }
gfCNCPoint4[22705] = {X 347.0031, Y 26.0886, Z -6.3333, A 0.000, B 0.000, C 0.000 }
gfCNCPoint4[22706] = {X 347.1054, Y 25.1822, Z -6.3333, A 0.000, B 0.000, C 0.000 }
gfCNCPoint4[22707] = {X 347.1011, Y 24.2701, Z -6.3333, A 0.000, B 0.000, C 0.000 }
gfCNCPoint4[22708] = {X 346.9902, Y 23.3647, Z -6.3333, A 0.000, B 0.000, C 0.000 }
gfCNCPoint4[22709] = {X 346.9489, Y 23.1616, Z -6.3333, A 0.000, B 0.000, C 0.000 }
gfCNCPoint4[22710] = {X 346.8828, Y 22.9651, Z -6.3333, A 0.000, B 0.000, C 0.000 }
gfCNCPoint4[22711] = {X 346.3962, Y 23.6864, Z -6.3333, A 0.000, B 0.000, C 0.000 }
gfCNCPoint4[22712] = {X 345.8671, Y 24.3770, Z -6.3333, A 0.000, B 0.000, C 0.000 }
gfCNCPoint4[22713] = {X 343.9666, Y 25.8427, Z -6.3333, A 0.000, B 0.000, C 0.000 }
gfCNCPoint4[22714] = {X 344.4658, Y 26.5398, Z -6.3333, A 0.000, B 0.000, C 0.000 }
gfCNCPoint4[22715] = {X 344.9143, Y 27.2706, Z -6.3333, A 0.000, B 0.000, C 0.000 }
gfCNCPoint4[22716] = {X 345.4664, Y 28.3742, Z -6.3333, A 0.000, B 0.000, C 0.000 }
gfCNCPoint4[22717] = {X 345.9030, Y 29.5284, Z -6.3333, A 0.000, B 0.000, C 0.000 }
gfCNCPoint4[22718] = {X 346.3596, Y 29.6189, Z -6.3333, A 0.000, B 0.000, C 0.000 }
gfCNCPoint4[22719] = {X 346.8248, Y 29.6329, Z -6.3333, A 0.000, B 0.000, C 0.000 }
gfCNCPoint4[22720] = {X 347.1176, Y 29.6178, Z -6.3333, A 0.000, B 0.000, C 0.000 }
gfCNCPoint4[22721] = {X 347.4785, Y 29.5389, Z -6.3333, A 0.000, B 0.000, C 0.000 }
gfCNCPoint4[22722] = {X 347.7949, Y 29.3482, Z -6.3333, A 0.000, B 0.000, C 0.000 }
gfCNCPoint4[22723] = {X 348.4747, Y 28.6289, Z -6.3333, A 0.000, B 0.000, C 0.000 }
gfCNCPoint4[22724] = {X 348.9850, Y 27.7807, Z -6.3333, A 0.000, B 0.000, C 0.000 }
gfCNCPoint4[22725] = {X 349.3021, Y 26.8432, Z -6.3333, A 0.000, B 0.000, C 0.000 }
gfCNCPoint4[22726] = {X 349.3366, Y 26.6704, Z -6.3333, A 0.000, B 0.000, C 0.000 }
gfCNCPoint4[22727] = {X 349.3680, Y 26.4971, Z -6.3333, A 0.000, B 0.000, C 0.000 }
gfCNCPoint4[22728] = {X 349.5013, Y 25.3232, Z -6.3333, A 0.000, B 0.000, C 0.000 }
gfCNCPoint4[22729] = {X 349.4978, Y 24.1417, Z -6.3333, A 0.000, B 0.000, C 0.000 }
gfCNCPoint4[22730] = {X 349.3575, Y 22.9685, Z -6.3333, A 0.000, B 0.000, C 0.000 }
gfCNCPoint4[22731] = {X 349.1796, Y 22.2565, Z -6.3333, A 0.000, B 0.000, C 0.000 }
gfCNCPoint4[22732] = {X 348.8770, Y 21.5879, Z -6.3333, A 0.000, B 0.000, C 0.000 }
gfCNCPoint4[22733] = {X 348.4595, Y 20.9843, Z -6.3333, A 0.000, B 0.000, C 0.000 }
gfCNCPoint4[22734] = {X 348.0919, Y 20.6603, Z -6.3333, A 0.000, B 0.000, C 0.000 }
gfCNCPoint4[22735] = {X 347.6346, Y 20.4840, Z -6.3333, A 0.000, B 0.000, C 0.000 }
gfCNCPoint4[22736] = {X 346.5775, Y 20.3825, Z -6.3333, A 0.000, B 0.000, C 0.000 }
gfCNCPoint4[22737] = {X 345.5202, Y 20.4823, Z -6.3333, A 0.000, B 0.000, C 0.000 }
gfCNCPoint4[22738] = {X 344.7180, Y 21.8933, Z -6.3333, A 0.000, B 0.000, C 0.000 }
gfCNCPoint4[22739] = {X 343.7339, Y 23.1840, Z -6.3333, A 0.000, B 0.000, C 0.000 }
gfCNCPoint4[22740] = {X 342.5857, Y 24.3311, Z -6.3333, A 0.000, B 0.000, C 0.000 }
gfCNCPoint4[22741] = {X 342.7815, Y 24.5198, Z -6.3333, A 0.000, B 0.000, C 0.000 }
gfCNCPoint4[22742] = {X 343.3984, Y 25.1594, Z -6.3333, A 0.000, B 0.000, C 0.000 }
gfCNCPoint4[22743] = {X 343.9666, Y 25.8427, Z -6.3333, A 0.000, B 0.000, C 0.000 }
gfCNCPoint4[22744] = {X 342.0661, Y 27.3083, Z -6.3333, A 0.000, B 0.000, C 0.000 }
gfCNCPoint4[22745] = {X 342.8614, Y 28.5165, Z -6.3333, A 0.000, B 0.000, C 0.000 }
gfCNCPoint4[22746] = {X 343.4678, Y 29.8297, Z -6.3333, A 0.000, B 0.000, C 0.000 }
gfCNCPoint4[22747] = {X 343.8717, Y 31.2186, Z -6.3333, A 0.000, B 0.000, C 0.000 }
gfCNCPoint4[22748] = {X 344.8343, Y 31.7006, Z -6.3333, A 0.000, B 0.000, C 0.000 }
gfCNCPoint4[22749] = {X 345.8753, Y 31.9748, Z -6.3333, A 0.000, B 0.000, C 0.000 }
gfCNCPoint4[22750] = {X 346.9505, Y 32.0297, Z -6.3333, A 0.000, B 0.000, C 0.000 }
gfCNCPoint4[22751] = {X 347.2417, Y 32.0146, Z -6.3333, A 0.000, B 0.000, C 0.000 }
gfCNCPoint4[22752] = {X 348.0010, Y 31.8915, Z -6.3333, A 0.000, B 0.000, C 0.000 }
gfCNCPoint4[22753] = {X 348.7156, Y 31.6070, Z -6.3333, A 0.000, B 0.000, C 0.000 }
gfCNCPoint4[22754] = {X 349.3518, Y 31.1747, Z -6.3333, A 0.000, B 0.000, C 0.000 }
gfCNCPoint4[22755] = {X 350.1527, Y 30.3712, Z -6.3333, A 0.000, B 0.000, C 0.000 }
gfCNCPoint4[22756] = {X 350.8133, Y 29.4489, Z -6.3333, A 0.000, B 0.000, C 0.000 }
gfCNCPoint4[22757] = {X 351.3163, Y 28.4321, Z -6.3333, A 0.000, B 0.000, C 0.000 }
gfCNCPoint4[22758] = {X 351.6485, Y 27.3474, Z -6.3333, A 0.000, B 0.000, C 0.000 }
gfCNCPoint4[22759] = {X 351.8770, Y 25.7621, Z -6.3333, A 0.000, B 0.000, C 0.000 }
gfCNCPoint4[22760] = {X 351.9023, Y 24.1607, Z -6.3333, A 0.000, B 0.000, C 0.000 }
gfCNCPoint4[22761] = {X 351.7240, Y 22.5690, Z -6.3333, A 0.000, B 0.000, C 0.000 }
gfCNCPoint4[22762] = {X 351.4420, Y 21.4555, Z -6.3333, A 0.000, B 0.000, C 0.000 }
gfCNCPoint4[22763] = {X 350.9677, Y 20.4093, Z -6.3333, A 0.000, B 0.000, C 0.000 }
gfCNCPoint4[22764] = {X 350.3161, Y 19.4634, Z -6.3333, A 0.000, B 0.000, C 0.000 }
gfCNCPoint4[22765] = {X 349.6855, Y 18.8476, Z -6.3333, A 0.000, B 0.000, C 0.000 }
gfCNCPoint4[22766] = {X 348.9297, Y 18.3941, Z -6.3333, A 0.000, B 0.000, C 0.000 }
gfCNCPoint4[22767] = {X 348.0895, Y 18.1275, Z -6.3333, A 0.000, B 0.000, C 0.000 }
gfCNCPoint4[22768] = {X 346.9970, Y 17.9937, Z -6.3333, A 0.000, B 0.000, C 0.000 }
gfCNCPoint4[22769] = {X 345.8965, Y 18.0111, Z -6.3333, A 0.000, B 0.000, C 0.000 }
gfCNCPoint4[22770] = {X 344.8087, Y 18.1794, Z -6.3333, A 0.000, B 0.000, C 0.000 }
gfCNCPoint4[22771] = {X 343.7543, Y 18.4953, Z -6.3333, A 0.000, B 0.000, C 0.000 }
gfCNCPoint4[22772] = {X 343.2662, Y 19.6257, Z -6.3333, A 0.000, B 0.000, C 0.000 }
gfCNCPoint4[22773] = {X 342.6386, Y 20.6850, Z -6.3333, A 0.000, B 0.000, C 0.000 }
gfCNCPoint4[22774] = {X 341.8815, Y 21.6560, Z -6.3333, A 0.000, B 0.000, C 0.000 }
gfCNCPoint4[22775] = {X 341.0073, Y 22.5231, Z -6.3333, A 0.000, B 0.000, C 0.000 }
gfCNCPoint4[22776] = {X 340.7217, Y 22.7629, Z -6.3333, A 0.000, B 0.000, C 0.000 }
gfCNCPoint4[22777] = {X 340.4270, Y 22.9916, Z -6.3333, A 0.000, B 0.000, C 0.000 }
gfCNCPoint4[22778] = {X 339.6615, Y 23.5549, Z -6.3333, A 0.000, B 0.000, C 0.000 }
gfCNCPoint4[22779] = {X 339.1299, Y 23.9121, Z -6.3333, A 0.000, B 0.000, C 0.000 }
gfCNCPoint4[22780] = {X 338.5759, Y 24.2333, Z -6.3333, A 0.000, B 0.000, C 0.000 }
gfCNCPoint4[22781] = {X 339.6077, Y 24.9034, Z -6.3333, A 0.000, B 0.000, C 0.000 }
gfCNCPoint4[22782] = {X 340.5462, Y 25.6989, Z -6.3333, A 0.000, B 0.000, C 0.000 }
gfCNCPoint4[22783] = {X 341.1165, Y 26.2483, Z -6.3333, A 0.000, B 0.000, C 0.000 }
gfCNCPoint4[22784] = {X 341.6108, Y 26.7608, Z -6.3333, A 0.000, B 0.000, C 0.000 }
gfCNCPoint4[22785] = {X 342.0661, Y 27.3083, Z -6.3333, A 0.000, B 0.000, C 0.000 }
gfCNCPoint4[22786] = {X 340.1656, Y 28.7740, Z -6.3333, A 0.000, B 0.000, C 0.000 }
gfCNCPoint4[22787] = {X 340.7330, Y 29.6278, Z -6.3333, A 0.000, B 0.000, C 0.000 }
gfCNCPoint4[22788] = {X 341.1747, Y 30.5529, Z -6.3333, A 0.000, B 0.000, C 0.000 }
gfCNCPoint4[22789] = {X 341.4822, Y 31.5308, Z -6.3333, A 0.000, B 0.000, C 0.000 }
gfCNCPoint4[22790] = {X 341.6492, Y 32.5422, Z -6.3333, A 0.000, B 0.000, C 0.000 }
gfCNCPoint4[22791] = {X 342.5908, Y 33.2482, Z -6.3333, A 0.000, B 0.000, C 0.000 }
gfCNCPoint4[22792] = {X 343.6298, Y 33.8008, Z -6.3333, A 0.000, B 0.000, C 0.000 }
gfCNCPoint4[22793] = {X 344.7416, Y 34.1868, Z -6.3333, A 0.000, B 0.000, C 0.000 }
gfCNCPoint4[22794] = {X 345.8995, Y 34.3970, Z -6.3333, A 0.000, B 0.000, C 0.000 }
gfCNCPoint4[22795] = {X 347.0761, Y 34.4264, Z -6.3333, A 0.000, B 0.000, C 0.000 }
gfCNCPoint4[22796] = {X 347.3657, Y 34.4114, Z -6.3333, A 0.000, B 0.000, C 0.000 }
gfCNCPoint4[22797] = {X 348.3266, Y 34.2824, Z -6.3333, A 0.000, B 0.000, C 0.000 }
gfCNCPoint4[22798] = {X 349.2536, Y 33.9986, Z -6.3333, A 0.000, B 0.000, C 0.000 }
gfCNCPoint4[22799] = {X 350.1221, Y 33.5677, Z -6.3333, A 0.000, B 0.000, C 0.000 }
gfCNCPoint4[22800] = {X 350.9088, Y 33.0011, Z -6.3333, A 0.000, B 0.000, C 0.000 }
gfCNCPoint4[22801] = {X 351.7849, Y 32.1500, Z -6.3333, A 0.000, B 0.000, C 0.000 }
gfCNCPoint4[22802] = {X 352.5432, Y 31.1926, Z -6.3333, A 0.000, B 0.000, C 0.000 }
gfCNCPoint4[22803] = {X 353.1711, Y 30.1449, Z -6.3333, A 0.000, B 0.000, C 0.000 }
